// TIA Portal project "BackUp" (V15)

(* hardware
DEVICE "S7-1200 station_1"  S7-1200 Station
   slot 0: "Rack_0"  S7-1200 Rack  Rack  V1.0
   slot 1: "PLC_1"  CPU 1214C DC/DC/DC  6ES7 214-1AG40-0XB0  V4.2
   slot 2: "DQ 8x24VDC _1"  SM 1222 DQ8 x 24VDC  6ES7 222-1BF32-0XB0  V2.0
*)

// ===== PLC "PLC_1"  CPU 1214C DC/DC/DC =====

VAR_GLOBAL   // PLC tag table "Tabla de variables estándar"
   "Ready" AT %I0.2 : Bool;
   "INP/ABSB0" AT %I0.0 : Bool;
   "ZSP/ABSB1" AT %I0.1 : Bool;
   "TLC/ABST Trans. Data Ready M" AT %I0.3 : Bool;
   "Alarm" AT %I0.4 : Bool;
   "SENSOR BOT LEFT" AT %I0.7 : Bool;
   "SENSOR BOT MID" AT %I0.6 : Bool;
   "SENSOR BOT RIGHT" AT %I0.5 : Bool;
   "SENSOR TOP LEFT" AT %I1.0 : Bool;
   "SENSOR TOP MID" AT %I1.1 : Bool;
   "SENSOR TOP RIGHT" AT %I1.2 : Bool;
   "SENSOR VERT TOP" AT %I1.3 : Bool;
   "SENSOR OPT. DOOR" AT %I1.5 : Bool;
   "SENSOR VERT BOT" AT %I1.4 : Bool;
   "Magnetic Brake" AT %Q8.6 : Bool;
   "Clear" AT %Q0.2 : Bool;
   "Axis_1_Pulse" AT %Q0.0 : Bool;
   "Axis_1_Direction" AT %Q0.1 : Bool;
   "PC/ABSM Transfer Mode" AT %Q0.3 : Bool;
   "TL/ABSR Request" AT %Q0.4 : Bool;
   "Son" AT %Q0.5 : Bool;
   "BOT. PNEU. ACT. RIGHT" AT %Q0.7 : Bool;
   "Lasers ON" AT %Q8.2 : Bool;
   "Lasers Zero 1" AT %Q8.3 : Bool;
   "Lasers Zero 2" AT %Q8.4 : Bool;
   "Lasers Zero 3" AT %Q8.5 : Bool;
   "PNEU. ACT. DOWN" AT %Q8.0 : Bool;
   "PNEU. ACT. UP" AT %Q8.1 : Bool;
   "BOT. PNEU. ACT. LEFT" AT %Q0.6 : Bool;
   "TOP. PNEU. ACT. LEFT" AT %Q1.0 : Bool;
   "TOP. PNEU. ACT. RIGHT" AT %Q1.1 : Bool;
   "Pilot Valve" AT %Q8.7 : Bool;
   "Magnetic Brake M" AT %M101.0 : Bool;
   "Set Home Axis" AT %M101.1 : Bool;
   "TL/ABSR Request M" AT %M0.3 : Bool;
   "PC/ABSM Transfer Mode M" AT %M0.2 : Bool;
   "Son M" AT %M101.2 : Bool;
   "INP/ABSB0 M" AT %M1.0 : Bool;
   "ZSP/ABSB1 M" AT %M1.1 : Bool;
   "TLC/ABST Trans. Data Ready" AT %M1.2 : Bool;
   "Step-0" AT %M5.0 : Bool;
   "Step-1" AT %M5.1 : Bool;
   "System_Byte" AT %MB3 : Byte;
   "FirstScan" AT %M3.0 : Bool;
   "DiagStatusUpdate" AT %M3.1 : Bool;
   "AlwaysTRUE" AT %M3.2 : Bool;
   "AlwaysFALSE" AT %M3.3 : Bool;
   "Step-2" AT %M5.2 : Bool;
   "Step-3" AT %M5.3 : Bool;
   "Step-4" AT %M5.4 : Bool;
   "Step-5" AT %M5.5 : Bool;
   "Step-6" AT %M5.6 : Bool;
   "Step-7" AT %M5.7 : Bool;
   "Step-8" AT %M6.0 : Bool;
   "Step-9" AT %M6.1 : Bool;
   "Step-10" AT %M6.2 : Bool;
   "Step-11" AT %M6.3 : Bool;
   "Step-12" AT %M6.4 : Bool;
   "Step-13" AT %M6.5 : Bool;
   "Step-14" AT %M6.6 : Bool;
   "Step-15" AT %M6.7 : Bool;
   "Step-16" AT %M7.0 : Bool;
   "Step-17" AT %M7.1 : Bool;
   "Step-18" AT %M7.2 : Bool;
   "Step-19" AT %M7.3 : Bool;
   "Step-20" AT %M7.4 : Bool;
   "Step-21" AT %M7.5 : Bool;
   "Step-22" AT %M7.6 : Bool;
   "Step-23" AT %M7.7 : Bool;
   "Step-24" AT %M8.0 : Bool;
   "Step-25" AT %M8.1 : Bool;
   "Step-26" AT %M8.2 : Bool;
   "Step-27" AT %M8.3 : Bool;
   "Step-28" AT %M8.4 : Bool;
   "Step-29" AT %M8.5 : Bool;
   "Step-30" AT %M8.6 : Bool;
   "Step-31" AT %M8.7 : Bool;
   "Step-32" AT %M9.0 : Bool;
   "Step-33" AT %M9.1 : Bool;
   "Step-34" AT %M9.2 : Bool;
   "Step-35" AT %M9.3 : Bool;
   "Step-36" AT %M9.4 : Bool;
   "Step-37" AT %M9.5 : Bool;
   "Step-38" AT %M9.6 : Bool;
   "Step-39" AT %M9.7 : Bool;
   "Step-40" AT %M10.0 : Bool;
   "Checksum OK" AT %M0.6 : Bool;
   "Step-41" AT %M10.1 : Bool;
   "Checksum M" AT %M0.7 : Bool;
   "Tranfer Mode Bit" AT %M1.3 : Bool;
   "Bit 25" AT %M11.0 : Bool;
   "Bit 26" AT %M11.1 : Bool;
   "Bit 27" AT %M11.2 : Bool;
   "Bit 28" AT %M11.3 : Bool;
   "Bit 29" AT %M11.4 : Bool;
   "Bit 30" AT %M11.5 : Bool;
   "Bit 31" AT %M11.6 : Bool;
   "Bit 32" AT %M11.7 : Bool;
   "Bit 17" AT %M12.0 : Bool;
   "Bit 18" AT %M12.1 : Bool;
   "Bit 19" AT %M12.2 : Bool;
   "Bit 20" AT %M12.3 : Bool;
   "Bit 21" AT %M12.4 : Bool;
   "Bit 22" AT %M12.5 : Bool;
   "Bit 23" AT %M12.6 : Bool;
   "Bit 24" AT %M12.7 : Bool;
   "Bit 9" AT %M13.0 : Bool;
   "Bit 10" AT %M13.1 : Bool;
   "Bit 11" AT %M13.2 : Bool;
   "Bit 12" AT %M13.3 : Bool;
   "Bit 13" AT %M13.4 : Bool;
   "Bit 14" AT %M13.5 : Bool;
   "Bit 15" AT %M13.6 : Bool;
   "Bit 16" AT %M13.7 : Bool;
   "Bit 1" AT %M14.0 : Bool;
   "Bit 2" AT %M14.1 : Bool;
   "Bit 3" AT %M14.2 : Bool;
   "Bit 4" AT %M14.3 : Bool;
   "Bit 5" AT %M14.4 : Bool;
   "Bit 6" AT %M14.5 : Bool;
   "Bit 7" AT %M14.6 : Bool;
   "Bit 8" AT %M14.7 : Bool;
   "Bit 1 Checksum" AT %M30.0 : Bool;
   "Bit 2 Checksum" AT %M30.1 : Bool;
   "Bit 3 Checksum" AT %M30.2 : Bool;
   "Bit 4 Checksum" AT %M30.3 : Bool;
   "Bit 5 Checksum" AT %M30.4 : Bool;
   "Bit 6 Checksum" AT %M30.5 : Bool;
   "ABS DoubleWord" AT %MD11 : DWord;
   "ABS DoubleInteger" AT %MD16 : DInt;
   "Checksum Byte" AT %MB30 : Byte;
   "Checksum Integer" AT %MW40 : Int;
   "Reset ABM Transfer" AT %M1.4 : Bool;
   "Step-42" AT %M10.2 : Bool;
   "Enable Axis" AT %M1.5 : Bool;
   "Move Absolute" AT %M101.3 : Bool;
   "Position" AT %MD42 : Real;
   "Velocity" AT %MD46 : Real;
   "Jog Back" AT %M101.4 : Bool;
   "Jog Forw" AT %M101.6 : Bool;
   "Jog" AT %M2.1 : Bool;
   "Home" AT %M2.2 : Bool;
   "Move Relative" AT %M101.7 : Bool;
   "BOT. PNEU. AUT. START" AT %M100.7 : Bool;
   "Lasers ON M" AT %M100.0 : Bool;
   "Lasers Zero 1 M" AT %M100.1 : Bool;
   "Lasers Zero 2 M" AT %M100.2 : Bool;
   "Lasers Zero 3 M" AT %M100.3 : Bool;
   "Home PLC" AT %M101.5 : Bool;
   "Home Done" AT %M138.0 : Bool;
   "Ramp Down" AT %MD50 : Real;
   "Ramp Up" AT %MD54 : Real;
   "Execute Ramp" AT %M103.0 : Bool;
   "Halt" AT %M103.1 : Bool;
   "BOT. PNEU. ACT. RIGHT M" AT %M100.5 : Bool;
   "BOT. PNEU. ACT. LEFT M" AT %M100.6 : Bool;
   "VELOCITY REAL" AT %MD700 : Real;
   "MB VELOCITY 2" AT %MW105 : UInt;
   "RAMP DOWN REAL" AT %MD704 : Real;
   "RAMP UP REAL" AT %MD708 : Real;
   "MB RAMP DOWN 2" AT %MW107 : UInt;
   "MB RAMP UP 2" AT %MW109 : UInt;
   "MB VELOCITY 1" AT %MW104 : UInt;
   "MB RAMP DOWN 1" AT %MW106 : UInt;
   "MB RAMP UP 1" AT %MW108 : UInt;
   "MB POSITION 1" AT %MW110 : UInt;
   "MB POSITION 2" AT %MW112 : UInt;
   "MB POSITION" AT %MD114 : DWord;
   "POSITION REAL" AT %MD118 : DInt;
   "Tag_4" AT %MW114 : UInt;
   "Tag_1" AT %MW116 : UInt;
   "PLC POSITION" AT %MD122 : Real;
   "PLC POS 1" AT %MW130 : UInt;
   "PLC POS 2" AT %MW132 : UInt;
   "PLC POS MULT" AT %MD126 : DInt;
   "PLC POS DW" AT %MD130 : DWord;
   "ABS POS" AT %MD134 : DWord;
   "Tag_2" AT %M500.0 : Bool;
   "Tag_3" AT %M500.1 : Bool;
   "Tag_5" AT %M500.2 : Bool;
   "Tag_6" AT %M400.0 : Bool;
   "HOME PNEU. ACT." AT %M100.4 : Bool;
   "Tag_8" AT %M400.1 : Bool;
   "Tag_9" AT %M500.6 : Bool;
   "Tag_10" AT %M500.4 : Bool;
   "Tag_11" AT %M500.5 : Bool;
   "Tag_12" AT %M500.3 : Bool;
   "Tag_13" AT %M501.0 : Bool;
   "Tag_14" AT %M501.1 : Bool;
   "Tag_15" AT %M501.2 : Bool;
   "Tag_16" AT %M501.3 : Bool;
   "Tag_17" AT %M501.4 : Bool;
   "Tag_18" AT %M501.5 : Bool;
   "Tag_19" AT %M501.6 : Bool;
   "Tag_20" AT %M501.7 : Bool;
   "Tag_21" AT %M502.0 : Bool;
   "Bot. Act. Mid. Pos." AT %M138.1 : Bool;
   "Bot. Act. Rig. Pos." AT %M138.2 : Bool;
   "TOP. PNEU. ACT. RIGHT M" AT %M103.2 : Bool;
   "TOP. PNEU. ACT. LEFT M" AT %M103.3 : Bool;
   "HEAD PNEU. ACT. DOWN" AT %M103.4 : Bool;
   "HEAD PNEU. ACT. UP" AT %M103.5 : Bool;
   "Tag_22" AT %M503.0 : Bool;
   "Tag_23" AT %M503.2 : Bool;
   "Tag_24" AT %M503.4 : Bool;
   "Tag_25" AT %M503.6 : Bool;
   "Tag_26" AT %M503.1 : Bool;
   "Tag_27" AT %M503.5 : Bool;
   "Tag_28" AT %M503.3 : Bool;
   "Tag_29" AT %M504.0 : Bool;
   "Tag_30" AT %M504.1 : Bool;
   "Tag_31" AT %M505.0 : Bool;
   "Tag_32" AT %M504.2 : Bool;
   "Tag_33" AT %M504.3 : Bool;
   "Tag_34" AT %M504.4 : Bool;
   "Tag_35" AT %M504.5 : Bool;
   "Tag_36" AT %M504.6 : Bool;
   "Tag_37" AT %M504.7 : Bool;
   "TOP. PNEU. AUT. START" AT %M103.6 : Bool;
   "Top Act. Mid. Pos." AT %M138.3 : Bool;
   "Top Act. Rig. Pos." AT %M138.4 : Bool;
   "Tag_7" AT %M506.0 : Bool;
   "Tag_38" AT %M506.1 : Bool;
   "Tag_39" AT %M506.2 : Bool;
   "Tag_40" AT %M506.3 : Bool;
   "Tag_41" AT %M506.4 : Bool;
   "HOME VERT. PNE. ACT." AT %M103.7 : Bool;
   "AUTO VERT. PNE. ACT." AT %M102.0 : Bool;
   "Tag_42" AT %M507.0 : Bool;
   "Tag_43" AT %M507.1 : Bool;
   "Tag_44" AT %M507.2 : Bool;
   "Tag_45" AT %M507.4 : Bool;
   "Tag_46" AT %M507.3 : Bool;
   "Tag_47" AT %M507.5 : Bool;
   "Door In Pos." AT %M138.5 : Bool;
   "Door Out Pos" AT %M138.6 : Bool;
   "Home Door" AT %M138.7 : Bool;
   "Tag_48" AT %M507.6 : Bool;
   "Pilot Valve M" AT %M102.1 : Bool;
   "Tag_49" AT %M503.7 : Bool;
   "Tag_50" AT %M500.7 : Bool;
   "Tag_51" AT %M505.1 : Bool;
   "Tag_52" AT %M502.1 : Bool;
END_VAR

DATA_BLOCK "MBConfig"   // DB13
{ S7_Optimized_Access := 'TRUE' }
VERSION : 0.1
   VAR
      CONNECT : TCON_IP_v4;
      NDR : Bool;
      DR : Bool;
      ERROR : Bool;
      STATE : Word;
   END_VAR
BEGIN
   CONNECT.InterfaceId := 64;
   CONNECT.ID := 1;
   CONNECT.ConnectionType := 11;
   CONNECT.RemoteAddress.ADDR[1] := 192;
   CONNECT.RemoteAddress.ADDR[2] := 168;
   CONNECT.RemoteAddress.ADDR[3] := 0;
   CONNECT.RemoteAddress.ADDR[4] := 101;
   CONNECT.LocalPort := 502;
END_DATA_BLOCK

DATA_BLOCK "BUFF"   // DB14
{ S7_Optimized_Access := 'TRUE' }
VERSION : 0.1
   VAR
      DATA : Array[0..100] of Word;
   END_VAR
BEGIN
END_DATA_BLOCK

DATA_BLOCK "RETAIN MEMORY"   // DB16
{ S7_Optimized_Access := 'TRUE' }
VERSION : 0.1
   VAR RETAIN
      SBLR : Bool;
      SBMR : Bool;
      SBRR : Bool;
      STLR : Bool;
      STMR : Bool;
      STRR : Bool;
      SVTR : Bool;
      SVBR : Bool;
   END_VAR
BEGIN
END_DATA_BLOCK

// folder: System blocks/Program resources

DATA_BLOCK "IEC_Timer_0_DB"   // DB2
{ S7_Optimized_Access := 'TRUE' }
AUTHOR : Simatic
FAMILY : IEC
NAME : IEC_TMR
VERSION : 1.0
// stored: InstanceOfName IEC_TIMER
"IEC_TIMER"
BEGIN
END_DATA_BLOCK

DATA_BLOCK "IEC_Timer_0_DB_1"   // DB3
{ S7_Optimized_Access := 'TRUE' }
AUTHOR : Simatic
FAMILY : IEC
NAME : IEC_TMR
VERSION : 1.0
// stored: InstanceOfName IEC_TIMER
"IEC_TIMER"
BEGIN
END_DATA_BLOCK

DATA_BLOCK "IEC_Timer_0_DB_3"   // DB5
{ S7_Optimized_Access := 'TRUE' }
AUTHOR : Simatic
FAMILY : IEC
NAME : IEC_TMR
VERSION : 1.0
// stored: InstanceOfName IEC_TIMER
"IEC_TIMER"
BEGIN
END_DATA_BLOCK

DATA_BLOCK "IEC_Timer_0_DB_2"   // DB15
{ S7_Optimized_Access := 'TRUE' }
AUTHOR : Simatic
FAMILY : IEC
NAME : IEC_TMR
VERSION : 1.0
// stored: InstanceOfName IEC_TIMER
"IEC_TIMER"
BEGIN
END_DATA_BLOCK

DATA_BLOCK "IEC_Timer_0_DB_4"   // DB17
{ S7_Optimized_Access := 'TRUE' }
AUTHOR : Simatic
FAMILY : IEC
NAME : IEC_TMR
VERSION : 1.0
// stored: InstanceOfName IEC_TIMER
"IEC_TIMER"
BEGIN
END_DATA_BLOCK

DATA_BLOCK "IEC_Timer_0_DB_5"   // DB18
{ S7_Optimized_Access := 'TRUE' }
AUTHOR : Simatic
FAMILY : IEC
NAME : IEC_TMR
VERSION : 1.0
// stored: InstanceOfName IEC_TIMER
"IEC_TIMER"
BEGIN
END_DATA_BLOCK

DATA_BLOCK "IEC_Timer_0_DB_6"   // DB19
{ S7_Optimized_Access := 'TRUE' }
AUTHOR : Simatic
FAMILY : IEC
NAME : IEC_TMR
VERSION : 1.0
// stored: InstanceOfName IEC_TIMER
"IEC_TIMER"
BEGIN
END_DATA_BLOCK

DATA_BLOCK "IEC_Timer_0_DB_7"   // DB20
{ S7_Optimized_Access := 'TRUE' }
AUTHOR : Simatic
FAMILY : IEC
NAME : IEC_TMR
VERSION : 1.0
// stored: InstanceOfName IEC_TIMER
"IEC_TIMER"
BEGIN
END_DATA_BLOCK

// folder: (top level)

DATA_BLOCK "Axis_1"   // DB1, Motion_DB
{ S7_Optimized_Access := 'TRUE' }
AUTHOR : SIMATIC
FAMILY : BasicMC
NAME : TO_PosAx
VERSION : 5.0
// stored: InstanceOfName TO_PositioningAxis
"TO_PositioningAxis"
BEGIN
   // Axis.LengthUnitNormalized.Distance = 1013
   // Axis.ReadyInput_AddressCU = %M3.2
   // Axis.OnlinePtoModeCU = 16#0000_0002
   // Axis.DirectionOutputEnabledCU = TRUE
   // Axis.SelectedChannel2EnumCU = %Q0.1
   // Axis.SelectedChannel1EnumCU = %Q0.0
   // Pulse.MinDeltaDeltaFrequencyCU = 0.004
   // Pulse.MaxDeltaDeltaFrequencyCU = 1.0E+10
   // Pulse.MinDeltaFrequencyCU = 0.005
   // Pulse.MaxDeltaFrequencyCU = 9.5E+9
   // Pulse.MinFrequencyCU = 1.0
   // Pulse.MaxFrequencyCU = 100000.0
   // Pulse.OutputSourceCU = 16#0000_0000
   // Axis.SelectPTO = 0
END_DATA_BLOCK

FUNCTION "GRAFCET ABS" : Void   // FC1, LAD
{ S7_Optimized_Access := 'TRUE' }
VERSION : 0.1
BEGIN

REGION Network 1
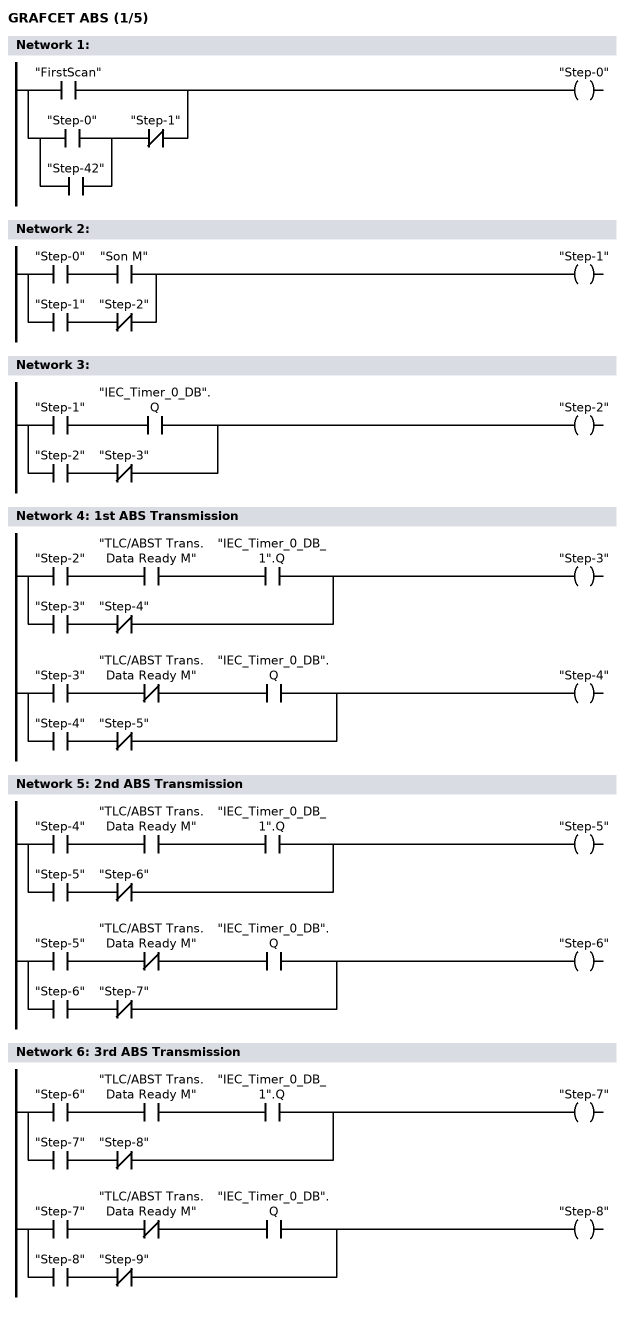
   RUNG wire#powerrail
      Contact( "FirstScan" )
      wire#w1
      Coil( "Step-0" )
   END_RUNG
   RUNG wire#powerrail
      Contact( "Step-0" )
      wire#w2
      I_Contact( "Step-1" )
   END_RUNG wire#w1
   RUNG wire#powerrail
      Contact( "Step-42" )
   END_RUNG wire#w2
   // the same network as SCL:
   "Step-0" := "FirstScan" OR (("Step-0" OR "Step-42") AND NOT "Step-1");
END_REGION

REGION Network 2
   RUNG wire#powerrail
      Contact( "Step-0" )
      Contact( "Son M" )
      wire#w1
      Coil( "Step-1" )
   END_RUNG
   RUNG wire#powerrail
      Contact( "Step-1" )
      I_Contact( "Step-2" )
   END_RUNG wire#w1
   // the same network as SCL:
   "Step-1" := ("Step-0" AND "Son M") OR ("Step-1" AND NOT "Step-2");
END_REGION

REGION Network 3
   RUNG wire#powerrail
      Contact( "Step-1" )
      Contact( "IEC_Timer_0_DB".Q )
      wire#w1
      Coil( "Step-2" )
   END_RUNG
   RUNG wire#powerrail
      Contact( "Step-2" )
      I_Contact( "Step-3" )
   END_RUNG wire#w1
   // the same network as SCL:
   "Step-2" := ("Step-1" AND "IEC_Timer_0_DB".Q) OR ("Step-2" AND NOT "Step-3");
END_REGION

REGION Network 4: 1st ABS Transmission
   RUNG wire#powerrail
      Contact( "Step-2" )
      Contact( "TLC/ABST Trans. Data Ready M" )
      Contact( "IEC_Timer_0_DB_1".Q )
      wire#w1
      Coil( "Step-3" )
   END_RUNG
   RUNG wire#powerrail
      Contact( "Step-3" )
      I_Contact( "Step-4" )
   END_RUNG wire#w1
   RUNG wire#powerrail
      Contact( "Step-3" )
      I_Contact( "TLC/ABST Trans. Data Ready M" )
      Contact( "IEC_Timer_0_DB".Q )
      wire#w2
      Coil( "Step-4" )
   END_RUNG
   RUNG wire#powerrail
      Contact( "Step-4" )
      I_Contact( "Step-5" )
   END_RUNG wire#w2
   // the same network as SCL:
   "Step-3" := ("Step-2" AND "TLC/ABST Trans. Data Ready M" AND "IEC_Timer_0_DB_1".Q) OR ("Step-3" AND NOT "Step-4");
   "Step-4" := ("Step-3" AND NOT "TLC/ABST Trans. Data Ready M" AND "IEC_Timer_0_DB".Q) OR ("Step-4" AND NOT "Step-5");
END_REGION

REGION Network 5: 2nd ABS Transmission
   RUNG wire#powerrail
      Contact( "Step-4" )
      Contact( "TLC/ABST Trans. Data Ready M" )
      Contact( "IEC_Timer_0_DB_1".Q )
      wire#w1
      Coil( "Step-5" )
   END_RUNG
   RUNG wire#powerrail
      Contact( "Step-5" )
      I_Contact( "Step-6" )
   END_RUNG wire#w1
   RUNG wire#powerrail
      Contact( "Step-5" )
      I_Contact( "TLC/ABST Trans. Data Ready M" )
      Contact( "IEC_Timer_0_DB".Q )
      wire#w2
      Coil( "Step-6" )
   END_RUNG
   RUNG wire#powerrail
      Contact( "Step-6" )
      I_Contact( "Step-7" )
   END_RUNG wire#w2
   // the same network as SCL:
   "Step-5" := ("Step-4" AND "TLC/ABST Trans. Data Ready M" AND "IEC_Timer_0_DB_1".Q) OR ("Step-5" AND NOT "Step-6");
   "Step-6" := ("Step-5" AND NOT "TLC/ABST Trans. Data Ready M" AND "IEC_Timer_0_DB".Q) OR ("Step-6" AND NOT "Step-7");
END_REGION

REGION Network 6: 3rd ABS Transmission
   RUNG wire#powerrail
      Contact( "Step-6" )
      Contact( "TLC/ABST Trans. Data Ready M" )
      Contact( "IEC_Timer_0_DB_1".Q )
      wire#w1
      Coil( "Step-7" )
   END_RUNG
   RUNG wire#powerrail
      Contact( "Step-7" )
      I_Contact( "Step-8" )
   END_RUNG wire#w1
   RUNG wire#powerrail
      Contact( "Step-7" )
      I_Contact( "TLC/ABST Trans. Data Ready M" )
      Contact( "IEC_Timer_0_DB".Q )
      wire#w2
      Coil( "Step-8" )
   END_RUNG
   RUNG wire#powerrail
      Contact( "Step-8" )
      I_Contact( "Step-9" )
   END_RUNG wire#w2
   // the same network as SCL:
   "Step-7" := ("Step-6" AND "TLC/ABST Trans. Data Ready M" AND "IEC_Timer_0_DB_1".Q) OR ("Step-7" AND NOT "Step-8");
   "Step-8" := ("Step-7" AND NOT "TLC/ABST Trans. Data Ready M" AND "IEC_Timer_0_DB".Q) OR ("Step-8" AND NOT "Step-9");
END_REGION

REGION Network 7: 4th ABS Transmission
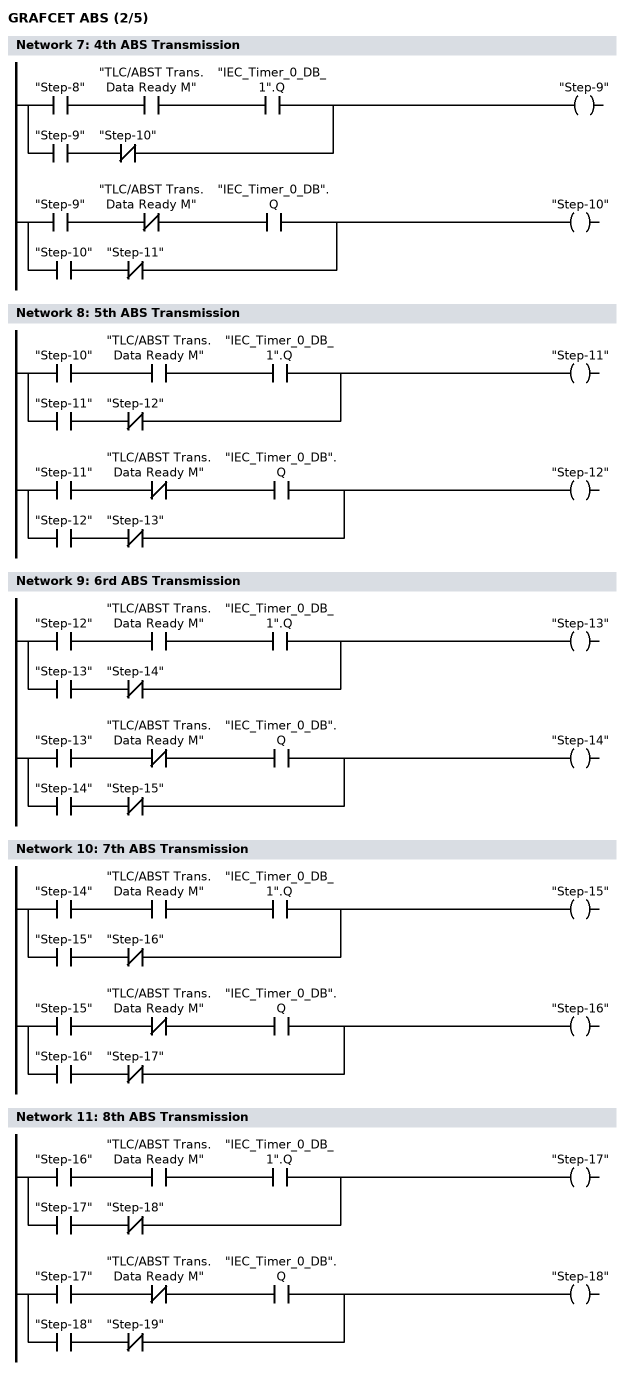
   RUNG wire#powerrail
      Contact( "Step-8" )
      Contact( "TLC/ABST Trans. Data Ready M" )
      Contact( "IEC_Timer_0_DB_1".Q )
      wire#w1
      Coil( "Step-9" )
   END_RUNG
   RUNG wire#powerrail
      Contact( "Step-9" )
      I_Contact( "Step-10" )
   END_RUNG wire#w1
   RUNG wire#powerrail
      Contact( "Step-9" )
      I_Contact( "TLC/ABST Trans. Data Ready M" )
      Contact( "IEC_Timer_0_DB".Q )
      wire#w2
      Coil( "Step-10" )
   END_RUNG
   RUNG wire#powerrail
      Contact( "Step-10" )
      I_Contact( "Step-11" )
   END_RUNG wire#w2
   // the same network as SCL:
   "Step-9" := ("Step-8" AND "TLC/ABST Trans. Data Ready M" AND "IEC_Timer_0_DB_1".Q) OR ("Step-9" AND NOT "Step-10");
   "Step-10" := ("Step-9" AND NOT "TLC/ABST Trans. Data Ready M" AND "IEC_Timer_0_DB".Q) OR ("Step-10" AND NOT "Step-11");
END_REGION

REGION Network 8: 5th ABS Transmission
   RUNG wire#powerrail
      Contact( "Step-10" )
      Contact( "TLC/ABST Trans. Data Ready M" )
      Contact( "IEC_Timer_0_DB_1".Q )
      wire#w1
      Coil( "Step-11" )
   END_RUNG
   RUNG wire#powerrail
      Contact( "Step-11" )
      I_Contact( "Step-12" )
   END_RUNG wire#w1
   RUNG wire#powerrail
      Contact( "Step-11" )
      I_Contact( "TLC/ABST Trans. Data Ready M" )
      Contact( "IEC_Timer_0_DB".Q )
      wire#w2
      Coil( "Step-12" )
   END_RUNG
   RUNG wire#powerrail
      Contact( "Step-12" )
      I_Contact( "Step-13" )
   END_RUNG wire#w2
   // the same network as SCL:
   "Step-11" := ("Step-10" AND "TLC/ABST Trans. Data Ready M" AND "IEC_Timer_0_DB_1".Q) OR ("Step-11" AND NOT "Step-12");
   "Step-12" := ("Step-11" AND NOT "TLC/ABST Trans. Data Ready M" AND "IEC_Timer_0_DB".Q) OR ("Step-12" AND NOT "Step-13");
END_REGION

REGION Network 9: 6rd ABS Transmission
   RUNG wire#powerrail
      Contact( "Step-12" )
      Contact( "TLC/ABST Trans. Data Ready M" )
      Contact( "IEC_Timer_0_DB_1".Q )
      wire#w1
      Coil( "Step-13" )
   END_RUNG
   RUNG wire#powerrail
      Contact( "Step-13" )
      I_Contact( "Step-14" )
   END_RUNG wire#w1
   RUNG wire#powerrail
      Contact( "Step-13" )
      I_Contact( "TLC/ABST Trans. Data Ready M" )
      Contact( "IEC_Timer_0_DB".Q )
      wire#w2
      Coil( "Step-14" )
   END_RUNG
   RUNG wire#powerrail
      Contact( "Step-14" )
      I_Contact( "Step-15" )
   END_RUNG wire#w2
   // the same network as SCL:
   "Step-13" := ("Step-12" AND "TLC/ABST Trans. Data Ready M" AND "IEC_Timer_0_DB_1".Q) OR ("Step-13" AND NOT "Step-14");
   "Step-14" := ("Step-13" AND NOT "TLC/ABST Trans. Data Ready M" AND "IEC_Timer_0_DB".Q) OR ("Step-14" AND NOT "Step-15");
END_REGION

REGION Network 10: 7th ABS Transmission
   RUNG wire#powerrail
      Contact( "Step-14" )
      Contact( "TLC/ABST Trans. Data Ready M" )
      Contact( "IEC_Timer_0_DB_1".Q )
      wire#w1
      Coil( "Step-15" )
   END_RUNG
   RUNG wire#powerrail
      Contact( "Step-15" )
      I_Contact( "Step-16" )
   END_RUNG wire#w1
   RUNG wire#powerrail
      Contact( "Step-15" )
      I_Contact( "TLC/ABST Trans. Data Ready M" )
      Contact( "IEC_Timer_0_DB".Q )
      wire#w2
      Coil( "Step-16" )
   END_RUNG
   RUNG wire#powerrail
      Contact( "Step-16" )
      I_Contact( "Step-17" )
   END_RUNG wire#w2
   // the same network as SCL:
   "Step-15" := ("Step-14" AND "TLC/ABST Trans. Data Ready M" AND "IEC_Timer_0_DB_1".Q) OR ("Step-15" AND NOT "Step-16");
   "Step-16" := ("Step-15" AND NOT "TLC/ABST Trans. Data Ready M" AND "IEC_Timer_0_DB".Q) OR ("Step-16" AND NOT "Step-17");
END_REGION

REGION Network 11: 8th ABS Transmission
   RUNG wire#powerrail
      Contact( "Step-16" )
      Contact( "TLC/ABST Trans. Data Ready M" )
      Contact( "IEC_Timer_0_DB_1".Q )
      wire#w1
      Coil( "Step-17" )
   END_RUNG
   RUNG wire#powerrail
      Contact( "Step-17" )
      I_Contact( "Step-18" )
   END_RUNG wire#w1
   RUNG wire#powerrail
      Contact( "Step-17" )
      I_Contact( "TLC/ABST Trans. Data Ready M" )
      Contact( "IEC_Timer_0_DB".Q )
      wire#w2
      Coil( "Step-18" )
   END_RUNG
   RUNG wire#powerrail
      Contact( "Step-18" )
      I_Contact( "Step-19" )
   END_RUNG wire#w2
   // the same network as SCL:
   "Step-17" := ("Step-16" AND "TLC/ABST Trans. Data Ready M" AND "IEC_Timer_0_DB_1".Q) OR ("Step-17" AND NOT "Step-18");
   "Step-18" := ("Step-17" AND NOT "TLC/ABST Trans. Data Ready M" AND "IEC_Timer_0_DB".Q) OR ("Step-18" AND NOT "Step-19");
END_REGION

REGION Network 12: 9th ABS Transmission
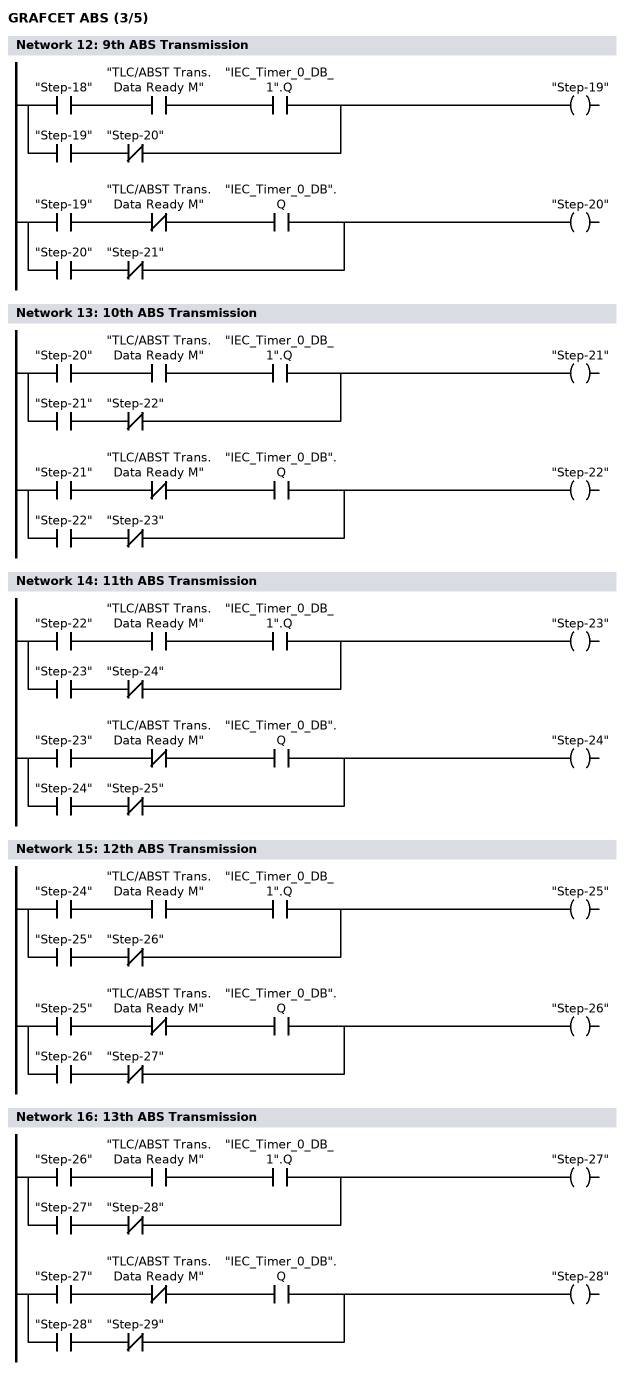
   RUNG wire#powerrail
      Contact( "Step-18" )
      Contact( "TLC/ABST Trans. Data Ready M" )
      Contact( "IEC_Timer_0_DB_1".Q )
      wire#w1
      Coil( "Step-19" )
   END_RUNG
   RUNG wire#powerrail
      Contact( "Step-19" )
      I_Contact( "Step-20" )
   END_RUNG wire#w1
   RUNG wire#powerrail
      Contact( "Step-19" )
      I_Contact( "TLC/ABST Trans. Data Ready M" )
      Contact( "IEC_Timer_0_DB".Q )
      wire#w2
      Coil( "Step-20" )
   END_RUNG
   RUNG wire#powerrail
      Contact( "Step-20" )
      I_Contact( "Step-21" )
   END_RUNG wire#w2
   // the same network as SCL:
   "Step-19" := ("Step-18" AND "TLC/ABST Trans. Data Ready M" AND "IEC_Timer_0_DB_1".Q) OR ("Step-19" AND NOT "Step-20");
   "Step-20" := ("Step-19" AND NOT "TLC/ABST Trans. Data Ready M" AND "IEC_Timer_0_DB".Q) OR ("Step-20" AND NOT "Step-21");
END_REGION

REGION Network 13: 10th ABS Transmission
   RUNG wire#powerrail
      Contact( "Step-20" )
      Contact( "TLC/ABST Trans. Data Ready M" )
      Contact( "IEC_Timer_0_DB_1".Q )
      wire#w1
      Coil( "Step-21" )
   END_RUNG
   RUNG wire#powerrail
      Contact( "Step-21" )
      I_Contact( "Step-22" )
   END_RUNG wire#w1
   RUNG wire#powerrail
      Contact( "Step-21" )
      I_Contact( "TLC/ABST Trans. Data Ready M" )
      Contact( "IEC_Timer_0_DB".Q )
      wire#w2
      Coil( "Step-22" )
   END_RUNG
   RUNG wire#powerrail
      Contact( "Step-22" )
      I_Contact( "Step-23" )
   END_RUNG wire#w2
   // the same network as SCL:
   "Step-21" := ("Step-20" AND "TLC/ABST Trans. Data Ready M" AND "IEC_Timer_0_DB_1".Q) OR ("Step-21" AND NOT "Step-22");
   "Step-22" := ("Step-21" AND NOT "TLC/ABST Trans. Data Ready M" AND "IEC_Timer_0_DB".Q) OR ("Step-22" AND NOT "Step-23");
END_REGION

REGION Network 14: 11th ABS Transmission
   RUNG wire#powerrail
      Contact( "Step-22" )
      Contact( "TLC/ABST Trans. Data Ready M" )
      Contact( "IEC_Timer_0_DB_1".Q )
      wire#w1
      Coil( "Step-23" )
   END_RUNG
   RUNG wire#powerrail
      Contact( "Step-23" )
      I_Contact( "Step-24" )
   END_RUNG wire#w1
   RUNG wire#powerrail
      Contact( "Step-23" )
      I_Contact( "TLC/ABST Trans. Data Ready M" )
      Contact( "IEC_Timer_0_DB".Q )
      wire#w2
      Coil( "Step-24" )
   END_RUNG
   RUNG wire#powerrail
      Contact( "Step-24" )
      I_Contact( "Step-25" )
   END_RUNG wire#w2
   // the same network as SCL:
   "Step-23" := ("Step-22" AND "TLC/ABST Trans. Data Ready M" AND "IEC_Timer_0_DB_1".Q) OR ("Step-23" AND NOT "Step-24");
   "Step-24" := ("Step-23" AND NOT "TLC/ABST Trans. Data Ready M" AND "IEC_Timer_0_DB".Q) OR ("Step-24" AND NOT "Step-25");
END_REGION

REGION Network 15: 12th ABS Transmission
   RUNG wire#powerrail
      Contact( "Step-24" )
      Contact( "TLC/ABST Trans. Data Ready M" )
      Contact( "IEC_Timer_0_DB_1".Q )
      wire#w1
      Coil( "Step-25" )
   END_RUNG
   RUNG wire#powerrail
      Contact( "Step-25" )
      I_Contact( "Step-26" )
   END_RUNG wire#w1
   RUNG wire#powerrail
      Contact( "Step-25" )
      I_Contact( "TLC/ABST Trans. Data Ready M" )
      Contact( "IEC_Timer_0_DB".Q )
      wire#w2
      Coil( "Step-26" )
   END_RUNG
   RUNG wire#powerrail
      Contact( "Step-26" )
      I_Contact( "Step-27" )
   END_RUNG wire#w2
   // the same network as SCL:
   "Step-25" := ("Step-24" AND "TLC/ABST Trans. Data Ready M" AND "IEC_Timer_0_DB_1".Q) OR ("Step-25" AND NOT "Step-26");
   "Step-26" := ("Step-25" AND NOT "TLC/ABST Trans. Data Ready M" AND "IEC_Timer_0_DB".Q) OR ("Step-26" AND NOT "Step-27");
END_REGION

REGION Network 16: 13th ABS Transmission
   RUNG wire#powerrail
      Contact( "Step-26" )
      Contact( "TLC/ABST Trans. Data Ready M" )
      Contact( "IEC_Timer_0_DB_1".Q )
      wire#w1
      Coil( "Step-27" )
   END_RUNG
   RUNG wire#powerrail
      Contact( "Step-27" )
      I_Contact( "Step-28" )
   END_RUNG wire#w1
   RUNG wire#powerrail
      Contact( "Step-27" )
      I_Contact( "TLC/ABST Trans. Data Ready M" )
      Contact( "IEC_Timer_0_DB".Q )
      wire#w2
      Coil( "Step-28" )
   END_RUNG
   RUNG wire#powerrail
      Contact( "Step-28" )
      I_Contact( "Step-29" )
   END_RUNG wire#w2
   // the same network as SCL:
   "Step-27" := ("Step-26" AND "TLC/ABST Trans. Data Ready M" AND "IEC_Timer_0_DB_1".Q) OR ("Step-27" AND NOT "Step-28");
   "Step-28" := ("Step-27" AND NOT "TLC/ABST Trans. Data Ready M" AND "IEC_Timer_0_DB".Q) OR ("Step-28" AND NOT "Step-29");
END_REGION

REGION Network 17: 14th ABS Transmission
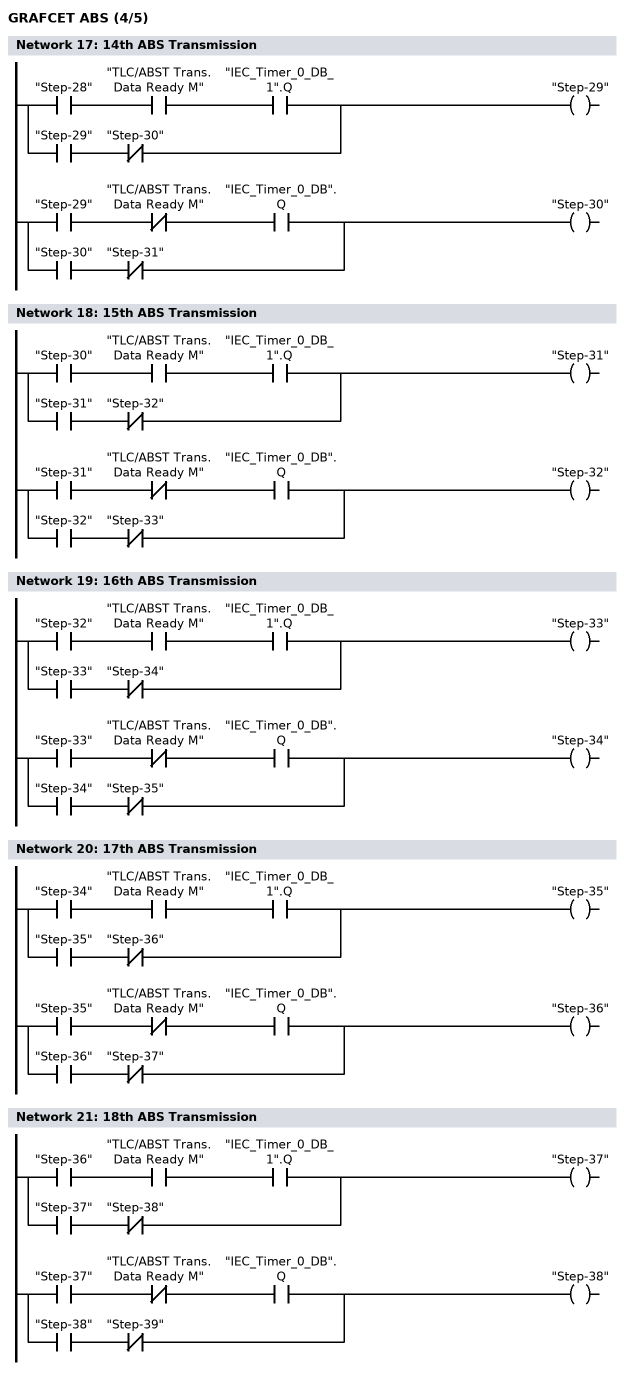
   RUNG wire#powerrail
      Contact( "Step-28" )
      Contact( "TLC/ABST Trans. Data Ready M" )
      Contact( "IEC_Timer_0_DB_1".Q )
      wire#w1
      Coil( "Step-29" )
   END_RUNG
   RUNG wire#powerrail
      Contact( "Step-29" )
      I_Contact( "Step-30" )
   END_RUNG wire#w1
   RUNG wire#powerrail
      Contact( "Step-29" )
      I_Contact( "TLC/ABST Trans. Data Ready M" )
      Contact( "IEC_Timer_0_DB".Q )
      wire#w2
      Coil( "Step-30" )
   END_RUNG
   RUNG wire#powerrail
      Contact( "Step-30" )
      I_Contact( "Step-31" )
   END_RUNG wire#w2
   // the same network as SCL:
   "Step-29" := ("Step-28" AND "TLC/ABST Trans. Data Ready M" AND "IEC_Timer_0_DB_1".Q) OR ("Step-29" AND NOT "Step-30");
   "Step-30" := ("Step-29" AND NOT "TLC/ABST Trans. Data Ready M" AND "IEC_Timer_0_DB".Q) OR ("Step-30" AND NOT "Step-31");
END_REGION

REGION Network 18: 15th ABS Transmission
   RUNG wire#powerrail
      Contact( "Step-30" )
      Contact( "TLC/ABST Trans. Data Ready M" )
      Contact( "IEC_Timer_0_DB_1".Q )
      wire#w1
      Coil( "Step-31" )
   END_RUNG
   RUNG wire#powerrail
      Contact( "Step-31" )
      I_Contact( "Step-32" )
   END_RUNG wire#w1
   RUNG wire#powerrail
      Contact( "Step-31" )
      I_Contact( "TLC/ABST Trans. Data Ready M" )
      Contact( "IEC_Timer_0_DB".Q )
      wire#w2
      Coil( "Step-32" )
   END_RUNG
   RUNG wire#powerrail
      Contact( "Step-32" )
      I_Contact( "Step-33" )
   END_RUNG wire#w2
   // the same network as SCL:
   "Step-31" := ("Step-30" AND "TLC/ABST Trans. Data Ready M" AND "IEC_Timer_0_DB_1".Q) OR ("Step-31" AND NOT "Step-32");
   "Step-32" := ("Step-31" AND NOT "TLC/ABST Trans. Data Ready M" AND "IEC_Timer_0_DB".Q) OR ("Step-32" AND NOT "Step-33");
END_REGION

REGION Network 19: 16th ABS Transmission
   RUNG wire#powerrail
      Contact( "Step-32" )
      Contact( "TLC/ABST Trans. Data Ready M" )
      Contact( "IEC_Timer_0_DB_1".Q )
      wire#w1
      Coil( "Step-33" )
   END_RUNG
   RUNG wire#powerrail
      Contact( "Step-33" )
      I_Contact( "Step-34" )
   END_RUNG wire#w1
   RUNG wire#powerrail
      Contact( "Step-33" )
      I_Contact( "TLC/ABST Trans. Data Ready M" )
      Contact( "IEC_Timer_0_DB".Q )
      wire#w2
      Coil( "Step-34" )
   END_RUNG
   RUNG wire#powerrail
      Contact( "Step-34" )
      I_Contact( "Step-35" )
   END_RUNG wire#w2
   // the same network as SCL:
   "Step-33" := ("Step-32" AND "TLC/ABST Trans. Data Ready M" AND "IEC_Timer_0_DB_1".Q) OR ("Step-33" AND NOT "Step-34");
   "Step-34" := ("Step-33" AND NOT "TLC/ABST Trans. Data Ready M" AND "IEC_Timer_0_DB".Q) OR ("Step-34" AND NOT "Step-35");
END_REGION

REGION Network 20: 17th ABS Transmission
   RUNG wire#powerrail
      Contact( "Step-34" )
      Contact( "TLC/ABST Trans. Data Ready M" )
      Contact( "IEC_Timer_0_DB_1".Q )
      wire#w1
      Coil( "Step-35" )
   END_RUNG
   RUNG wire#powerrail
      Contact( "Step-35" )
      I_Contact( "Step-36" )
   END_RUNG wire#w1
   RUNG wire#powerrail
      Contact( "Step-35" )
      I_Contact( "TLC/ABST Trans. Data Ready M" )
      Contact( "IEC_Timer_0_DB".Q )
      wire#w2
      Coil( "Step-36" )
   END_RUNG
   RUNG wire#powerrail
      Contact( "Step-36" )
      I_Contact( "Step-37" )
   END_RUNG wire#w2
   // the same network as SCL:
   "Step-35" := ("Step-34" AND "TLC/ABST Trans. Data Ready M" AND "IEC_Timer_0_DB_1".Q) OR ("Step-35" AND NOT "Step-36");
   "Step-36" := ("Step-35" AND NOT "TLC/ABST Trans. Data Ready M" AND "IEC_Timer_0_DB".Q) OR ("Step-36" AND NOT "Step-37");
END_REGION

REGION Network 21: 18th ABS Transmission
   RUNG wire#powerrail
      Contact( "Step-36" )
      Contact( "TLC/ABST Trans. Data Ready M" )
      Contact( "IEC_Timer_0_DB_1".Q )
      wire#w1
      Coil( "Step-37" )
   END_RUNG
   RUNG wire#powerrail
      Contact( "Step-37" )
      I_Contact( "Step-38" )
   END_RUNG wire#w1
   RUNG wire#powerrail
      Contact( "Step-37" )
      I_Contact( "TLC/ABST Trans. Data Ready M" )
      Contact( "IEC_Timer_0_DB".Q )
      wire#w2
      Coil( "Step-38" )
   END_RUNG
   RUNG wire#powerrail
      Contact( "Step-38" )
      I_Contact( "Step-39" )
   END_RUNG wire#w2
   // the same network as SCL:
   "Step-37" := ("Step-36" AND "TLC/ABST Trans. Data Ready M" AND "IEC_Timer_0_DB_1".Q) OR ("Step-37" AND NOT "Step-38");
   "Step-38" := ("Step-37" AND NOT "TLC/ABST Trans. Data Ready M" AND "IEC_Timer_0_DB".Q) OR ("Step-38" AND NOT "Step-39");
END_REGION

REGION Network 22: 19th ABS Transmission
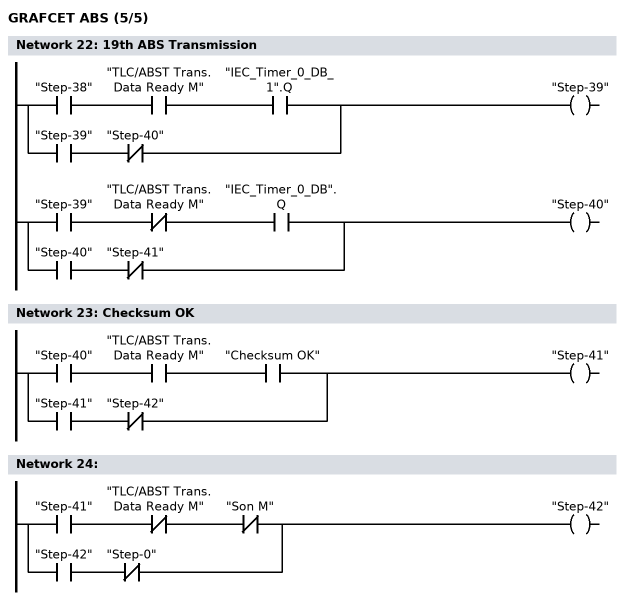
   RUNG wire#powerrail
      Contact( "Step-38" )
      Contact( "TLC/ABST Trans. Data Ready M" )
      Contact( "IEC_Timer_0_DB_1".Q )
      wire#w1
      Coil( "Step-39" )
   END_RUNG
   RUNG wire#powerrail
      Contact( "Step-39" )
      I_Contact( "Step-40" )
   END_RUNG wire#w1
   RUNG wire#powerrail
      Contact( "Step-39" )
      I_Contact( "TLC/ABST Trans. Data Ready M" )
      Contact( "IEC_Timer_0_DB".Q )
      wire#w2
      Coil( "Step-40" )
   END_RUNG
   RUNG wire#powerrail
      Contact( "Step-40" )
      I_Contact( "Step-41" )
   END_RUNG wire#w2
   // the same network as SCL:
   "Step-39" := ("Step-38" AND "TLC/ABST Trans. Data Ready M" AND "IEC_Timer_0_DB_1".Q) OR ("Step-39" AND NOT "Step-40");
   "Step-40" := ("Step-39" AND NOT "TLC/ABST Trans. Data Ready M" AND "IEC_Timer_0_DB".Q) OR ("Step-40" AND NOT "Step-41");
END_REGION

REGION Network 23: Checksum OK
   RUNG wire#powerrail
      Contact( "Step-40" )
      Contact( "TLC/ABST Trans. Data Ready M" )
      Contact( "Checksum OK" )
      wire#w1
      Coil( "Step-41" )
   END_RUNG
   RUNG wire#powerrail
      Contact( "Step-41" )
      I_Contact( "Step-42" )
   END_RUNG wire#w1
   // the same network as SCL:
   "Step-41" := ("Step-40" AND "TLC/ABST Trans. Data Ready M" AND "Checksum OK") OR ("Step-41" AND NOT "Step-42");
END_REGION

REGION Network 24
   RUNG wire#powerrail
      Contact( "Step-41" )
      I_Contact( "TLC/ABST Trans. Data Ready M" )
      I_Contact( "Son M" )
      wire#w1
      Coil( "Step-42" )
   END_RUNG
   RUNG wire#powerrail
      Contact( "Step-42" )
      I_Contact( "Step-0" )
   END_RUNG wire#w1
   // the same network as SCL:
   "Step-42" := ("Step-41" AND NOT "TLC/ABST Trans. Data Ready M" AND NOT "Son M") OR ("Step-42" AND NOT "Step-0");
END_REGION
END_FUNCTION

FUNCTION "OUTPUT GRAFCET ABS" : Void   // FC2, LAD
{ S7_Optimized_Access := 'TRUE' }
VERSION : 0.1
   VAR_TEMP   // added for the SCL form of the ladder/FBD networks
      _w1 : Bool;
   END_VAR
BEGIN

REGION Network 1
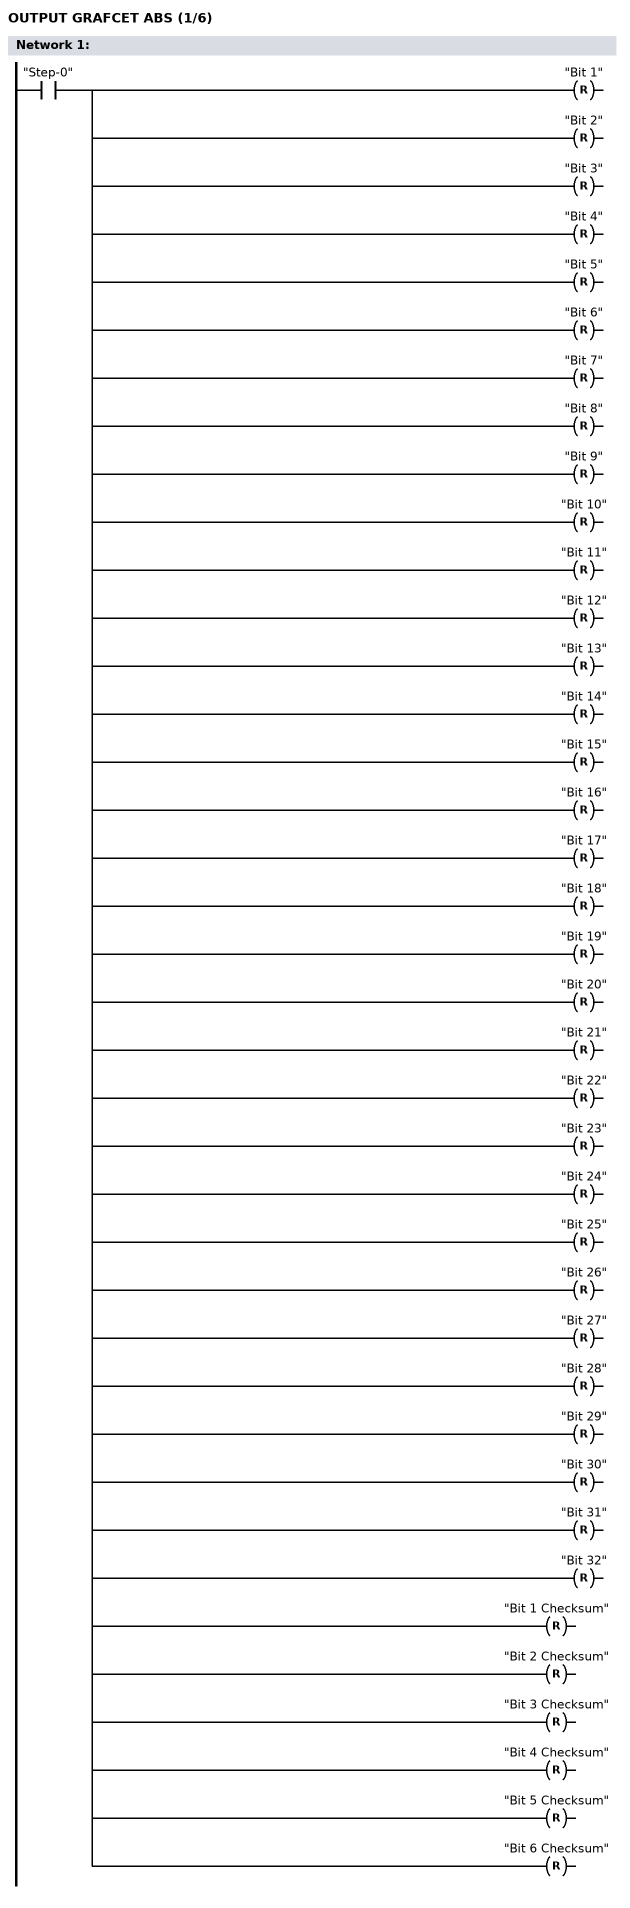
   RUNG wire#powerrail
      Contact( "Step-0" )
      wire#w1
      R_Coil( "Bit 1" )
   END_RUNG
   RUNG wire#w1
      R_Coil( "Bit 2" )
   END_RUNG
   RUNG wire#w1
      R_Coil( "Bit 3" )
   END_RUNG
   RUNG wire#w1
      R_Coil( "Bit 4" )
   END_RUNG
   RUNG wire#w1
      R_Coil( "Bit 5" )
   END_RUNG
   RUNG wire#w1
      R_Coil( "Bit 6" )
   END_RUNG
   RUNG wire#w1
      R_Coil( "Bit 7" )
   END_RUNG
   RUNG wire#w1
      R_Coil( "Bit 8" )
   END_RUNG
   RUNG wire#w1
      R_Coil( "Bit 9" )
   END_RUNG
   RUNG wire#w1
      R_Coil( "Bit 10" )
   END_RUNG
   RUNG wire#w1
      R_Coil( "Bit 11" )
   END_RUNG
   RUNG wire#w1
      R_Coil( "Bit 12" )
   END_RUNG
   RUNG wire#w1
      R_Coil( "Bit 13" )
   END_RUNG
   RUNG wire#w1
      R_Coil( "Bit 14" )
   END_RUNG
   RUNG wire#w1
      R_Coil( "Bit 15" )
   END_RUNG
   RUNG wire#w1
      R_Coil( "Bit 16" )
   END_RUNG
   RUNG wire#w1
      R_Coil( "Bit 17" )
   END_RUNG
   RUNG wire#w1
      R_Coil( "Bit 18" )
   END_RUNG
   RUNG wire#w1
      R_Coil( "Bit 19" )
   END_RUNG
   RUNG wire#w1
      R_Coil( "Bit 20" )
   END_RUNG
   RUNG wire#w1
      R_Coil( "Bit 21" )
   END_RUNG
   RUNG wire#w1
      R_Coil( "Bit 22" )
   END_RUNG
   RUNG wire#w1
      R_Coil( "Bit 23" )
   END_RUNG
   RUNG wire#w1
      R_Coil( "Bit 24" )
   END_RUNG
   RUNG wire#w1
      R_Coil( "Bit 25" )
   END_RUNG
   RUNG wire#w1
      R_Coil( "Bit 26" )
   END_RUNG
   RUNG wire#w1
      R_Coil( "Bit 27" )
   END_RUNG
   RUNG wire#w1
      R_Coil( "Bit 28" )
   END_RUNG
   RUNG wire#w1
      R_Coil( "Bit 29" )
   END_RUNG
   RUNG wire#w1
      R_Coil( "Bit 30" )
   END_RUNG
   RUNG wire#w1
      R_Coil( "Bit 31" )
   END_RUNG
   RUNG wire#w1
      R_Coil( "Bit 32" )
   END_RUNG
   RUNG wire#w1
      R_Coil( "Bit 1 Checksum" )
   END_RUNG
   RUNG wire#w1
      R_Coil( "Bit 2 Checksum" )
   END_RUNG
   RUNG wire#w1
      R_Coil( "Bit 3 Checksum" )
   END_RUNG
   RUNG wire#w1
      R_Coil( "Bit 4 Checksum" )
   END_RUNG
   RUNG wire#w1
      R_Coil( "Bit 5 Checksum" )
   END_RUNG
   RUNG wire#w1
      R_Coil( "Bit 6 Checksum" )
   END_RUNG
   // the same network as SCL:
   IF "Step-0" THEN
       "Bit 1" := FALSE;
       "Bit 2" := FALSE;
       "Bit 3" := FALSE;
       "Bit 4" := FALSE;
       "Bit 5" := FALSE;
       "Bit 6" := FALSE;
       "Bit 7" := FALSE;
       "Bit 8" := FALSE;
       "Bit 9" := FALSE;
       "Bit 10" := FALSE;
       "Bit 11" := FALSE;
       "Bit 12" := FALSE;
       "Bit 13" := FALSE;
       "Bit 14" := FALSE;
       "Bit 15" := FALSE;
       "Bit 16" := FALSE;
       "Bit 17" := FALSE;
       "Bit 18" := FALSE;
       "Bit 19" := FALSE;
       "Bit 20" := FALSE;
       "Bit 21" := FALSE;
       "Bit 22" := FALSE;
       "Bit 23" := FALSE;
       "Bit 24" := FALSE;
       "Bit 25" := FALSE;
       "Bit 26" := FALSE;
       "Bit 27" := FALSE;
       "Bit 28" := FALSE;
       "Bit 29" := FALSE;
       "Bit 30" := FALSE;
       "Bit 31" := FALSE;
       "Bit 32" := FALSE;
       "Bit 1 Checksum" := FALSE;
       "Bit 2 Checksum" := FALSE;
       "Bit 3 Checksum" := FALSE;
       "Bit 4 Checksum" := FALSE;
       "Bit 5 Checksum" := FALSE;
       "Bit 6 Checksum" := FALSE;
   END_IF;
END_REGION

REGION Network 2: Step-1
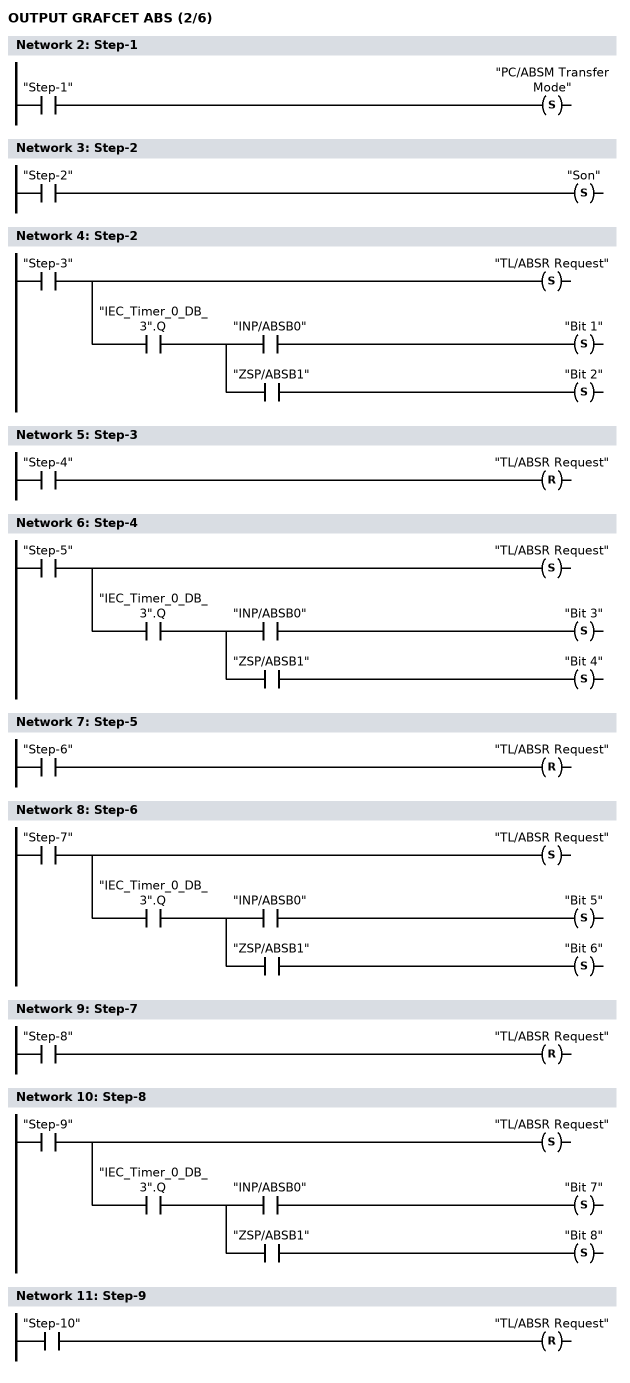
   RUNG wire#powerrail
      Contact( "Step-1" )
      S_Coil( "PC/ABSM Transfer Mode" )
   END_RUNG
   // the same network as SCL:
   IF "Step-1" THEN "PC/ABSM Transfer Mode" := TRUE; END_IF;
END_REGION

REGION Network 3: Step-2
   RUNG wire#powerrail
      Contact( "Step-2" )
      S_Coil( "Son" )
   END_RUNG
   // the same network as SCL:
   IF "Step-2" THEN "Son" := TRUE; END_IF;
END_REGION

REGION Network 4: Step-2
   RUNG wire#powerrail
      Contact( "Step-3" )
      wire#w1
      S_Coil( "TL/ABSR Request" )
   END_RUNG
   RUNG wire#w1
      Contact( "IEC_Timer_0_DB_3".Q )
      wire#w2
      Contact( "INP/ABSB0" )
      S_Coil( "Bit 1" )
   END_RUNG
   RUNG wire#w2
      Contact( "ZSP/ABSB1" )
      S_Coil( "Bit 2" )
   END_RUNG
   // the same network as SCL:
   IF "Step-3" THEN "TL/ABSR Request" := TRUE; END_IF;
   #_w1 := "Step-3" AND "IEC_Timer_0_DB_3".Q;
   IF #_w1 AND "INP/ABSB0" THEN "Bit 1" := TRUE; END_IF;
   IF #_w1 AND "ZSP/ABSB1" THEN "Bit 2" := TRUE; END_IF;
END_REGION

REGION Network 5: Step-3
   RUNG wire#powerrail
      Contact( "Step-4" )
      R_Coil( "TL/ABSR Request" )
   END_RUNG
   // the same network as SCL:
   IF "Step-4" THEN "TL/ABSR Request" := FALSE; END_IF;
END_REGION

REGION Network 6: Step-4
   RUNG wire#powerrail
      Contact( "Step-5" )
      wire#w1
      S_Coil( "TL/ABSR Request" )
   END_RUNG
   RUNG wire#w1
      Contact( "IEC_Timer_0_DB_3".Q )
      wire#w2
      Contact( "INP/ABSB0" )
      S_Coil( "Bit 3" )
   END_RUNG
   RUNG wire#w2
      Contact( "ZSP/ABSB1" )
      S_Coil( "Bit 4" )
   END_RUNG
   // the same network as SCL:
   IF "Step-5" THEN "TL/ABSR Request" := TRUE; END_IF;
   #_w1 := "Step-5" AND "IEC_Timer_0_DB_3".Q;
   IF #_w1 AND "INP/ABSB0" THEN "Bit 3" := TRUE; END_IF;
   IF #_w1 AND "ZSP/ABSB1" THEN "Bit 4" := TRUE; END_IF;
END_REGION

REGION Network 7: Step-5
   RUNG wire#powerrail
      Contact( "Step-6" )
      R_Coil( "TL/ABSR Request" )
   END_RUNG
   // the same network as SCL:
   IF "Step-6" THEN "TL/ABSR Request" := FALSE; END_IF;
END_REGION

REGION Network 8: Step-6
   RUNG wire#powerrail
      Contact( "Step-7" )
      wire#w1
      S_Coil( "TL/ABSR Request" )
   END_RUNG
   RUNG wire#w1
      Contact( "IEC_Timer_0_DB_3".Q )
      wire#w2
      Contact( "INP/ABSB0" )
      S_Coil( "Bit 5" )
   END_RUNG
   RUNG wire#w2
      Contact( "ZSP/ABSB1" )
      S_Coil( "Bit 6" )
   END_RUNG
   // the same network as SCL:
   IF "Step-7" THEN "TL/ABSR Request" := TRUE; END_IF;
   #_w1 := "Step-7" AND "IEC_Timer_0_DB_3".Q;
   IF #_w1 AND "INP/ABSB0" THEN "Bit 5" := TRUE; END_IF;
   IF #_w1 AND "ZSP/ABSB1" THEN "Bit 6" := TRUE; END_IF;
END_REGION

REGION Network 9: Step-7
   RUNG wire#powerrail
      Contact( "Step-8" )
      R_Coil( "TL/ABSR Request" )
   END_RUNG
   // the same network as SCL:
   IF "Step-8" THEN "TL/ABSR Request" := FALSE; END_IF;
END_REGION

REGION Network 10: Step-8
   RUNG wire#powerrail
      Contact( "Step-9" )
      wire#w1
      S_Coil( "TL/ABSR Request" )
   END_RUNG
   RUNG wire#w1
      Contact( "IEC_Timer_0_DB_3".Q )
      wire#w2
      Contact( "INP/ABSB0" )
      S_Coil( "Bit 7" )
   END_RUNG
   RUNG wire#w2
      Contact( "ZSP/ABSB1" )
      S_Coil( "Bit 8" )
   END_RUNG
   // the same network as SCL:
   IF "Step-9" THEN "TL/ABSR Request" := TRUE; END_IF;
   #_w1 := "Step-9" AND "IEC_Timer_0_DB_3".Q;
   IF #_w1 AND "INP/ABSB0" THEN "Bit 7" := TRUE; END_IF;
   IF #_w1 AND "ZSP/ABSB1" THEN "Bit 8" := TRUE; END_IF;
END_REGION

REGION Network 11: Step-9
   RUNG wire#powerrail
      Contact( "Step-10" )
      R_Coil( "TL/ABSR Request" )
   END_RUNG
   // the same network as SCL:
   IF "Step-10" THEN "TL/ABSR Request" := FALSE; END_IF;
END_REGION

REGION Network 12: Step-10
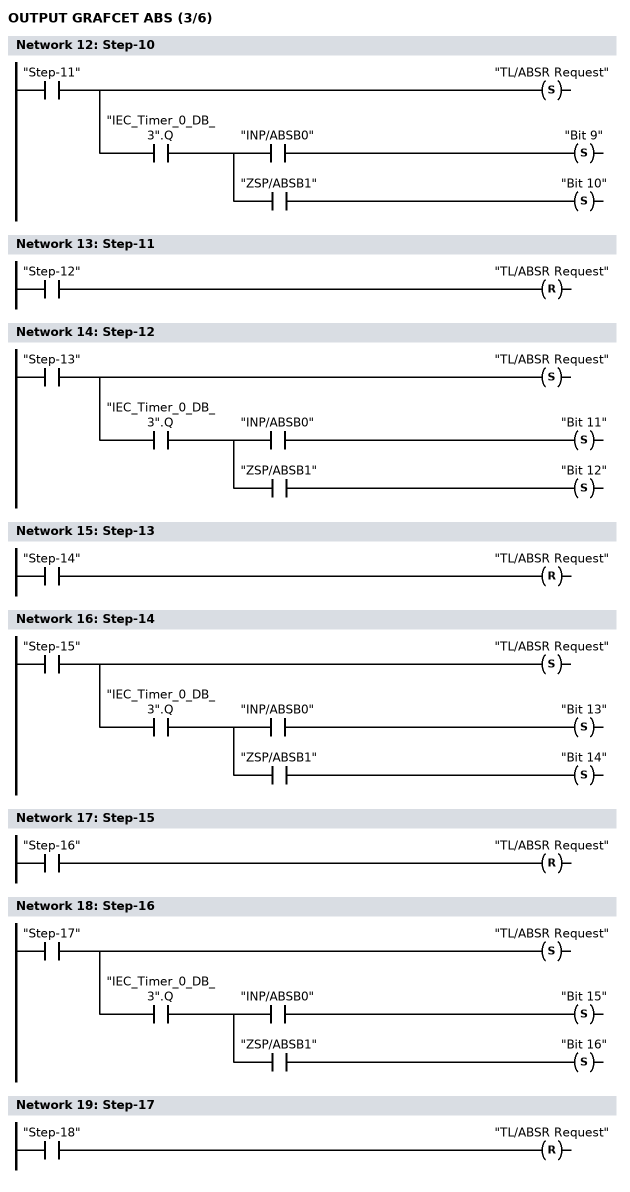
   RUNG wire#powerrail
      Contact( "Step-11" )
      wire#w1
      S_Coil( "TL/ABSR Request" )
   END_RUNG
   RUNG wire#w1
      Contact( "IEC_Timer_0_DB_3".Q )
      wire#w2
      Contact( "INP/ABSB0" )
      S_Coil( "Bit 9" )
   END_RUNG
   RUNG wire#w2
      Contact( "ZSP/ABSB1" )
      S_Coil( "Bit 10" )
   END_RUNG
   // the same network as SCL:
   IF "Step-11" THEN "TL/ABSR Request" := TRUE; END_IF;
   #_w1 := "Step-11" AND "IEC_Timer_0_DB_3".Q;
   IF #_w1 AND "INP/ABSB0" THEN "Bit 9" := TRUE; END_IF;
   IF #_w1 AND "ZSP/ABSB1" THEN "Bit 10" := TRUE; END_IF;
END_REGION

REGION Network 13: Step-11
   RUNG wire#powerrail
      Contact( "Step-12" )
      R_Coil( "TL/ABSR Request" )
   END_RUNG
   // the same network as SCL:
   IF "Step-12" THEN "TL/ABSR Request" := FALSE; END_IF;
END_REGION

REGION Network 14: Step-12
   RUNG wire#powerrail
      Contact( "Step-13" )
      wire#w1
      S_Coil( "TL/ABSR Request" )
   END_RUNG
   RUNG wire#w1
      Contact( "IEC_Timer_0_DB_3".Q )
      wire#w2
      Contact( "INP/ABSB0" )
      S_Coil( "Bit 11" )
   END_RUNG
   RUNG wire#w2
      Contact( "ZSP/ABSB1" )
      S_Coil( "Bit 12" )
   END_RUNG
   // the same network as SCL:
   IF "Step-13" THEN "TL/ABSR Request" := TRUE; END_IF;
   #_w1 := "Step-13" AND "IEC_Timer_0_DB_3".Q;
   IF #_w1 AND "INP/ABSB0" THEN "Bit 11" := TRUE; END_IF;
   IF #_w1 AND "ZSP/ABSB1" THEN "Bit 12" := TRUE; END_IF;
END_REGION

REGION Network 15: Step-13
   RUNG wire#powerrail
      Contact( "Step-14" )
      R_Coil( "TL/ABSR Request" )
   END_RUNG
   // the same network as SCL:
   IF "Step-14" THEN "TL/ABSR Request" := FALSE; END_IF;
END_REGION

REGION Network 16: Step-14
   RUNG wire#powerrail
      Contact( "Step-15" )
      wire#w1
      S_Coil( "TL/ABSR Request" )
   END_RUNG
   RUNG wire#w1
      Contact( "IEC_Timer_0_DB_3".Q )
      wire#w2
      Contact( "INP/ABSB0" )
      S_Coil( "Bit 13" )
   END_RUNG
   RUNG wire#w2
      Contact( "ZSP/ABSB1" )
      S_Coil( "Bit 14" )
   END_RUNG
   // the same network as SCL:
   IF "Step-15" THEN "TL/ABSR Request" := TRUE; END_IF;
   #_w1 := "Step-15" AND "IEC_Timer_0_DB_3".Q;
   IF #_w1 AND "INP/ABSB0" THEN "Bit 13" := TRUE; END_IF;
   IF #_w1 AND "ZSP/ABSB1" THEN "Bit 14" := TRUE; END_IF;
END_REGION

REGION Network 17: Step-15
   RUNG wire#powerrail
      Contact( "Step-16" )
      R_Coil( "TL/ABSR Request" )
   END_RUNG
   // the same network as SCL:
   IF "Step-16" THEN "TL/ABSR Request" := FALSE; END_IF;
END_REGION

REGION Network 18: Step-16
   RUNG wire#powerrail
      Contact( "Step-17" )
      wire#w1
      S_Coil( "TL/ABSR Request" )
   END_RUNG
   RUNG wire#w1
      Contact( "IEC_Timer_0_DB_3".Q )
      wire#w2
      Contact( "INP/ABSB0" )
      S_Coil( "Bit 15" )
   END_RUNG
   RUNG wire#w2
      Contact( "ZSP/ABSB1" )
      S_Coil( "Bit 16" )
   END_RUNG
   // the same network as SCL:
   IF "Step-17" THEN "TL/ABSR Request" := TRUE; END_IF;
   #_w1 := "Step-17" AND "IEC_Timer_0_DB_3".Q;
   IF #_w1 AND "INP/ABSB0" THEN "Bit 15" := TRUE; END_IF;
   IF #_w1 AND "ZSP/ABSB1" THEN "Bit 16" := TRUE; END_IF;
END_REGION

REGION Network 19: Step-17
   RUNG wire#powerrail
      Contact( "Step-18" )
      R_Coil( "TL/ABSR Request" )
   END_RUNG
   // the same network as SCL:
   IF "Step-18" THEN "TL/ABSR Request" := FALSE; END_IF;
END_REGION

REGION Network 20: Step-18
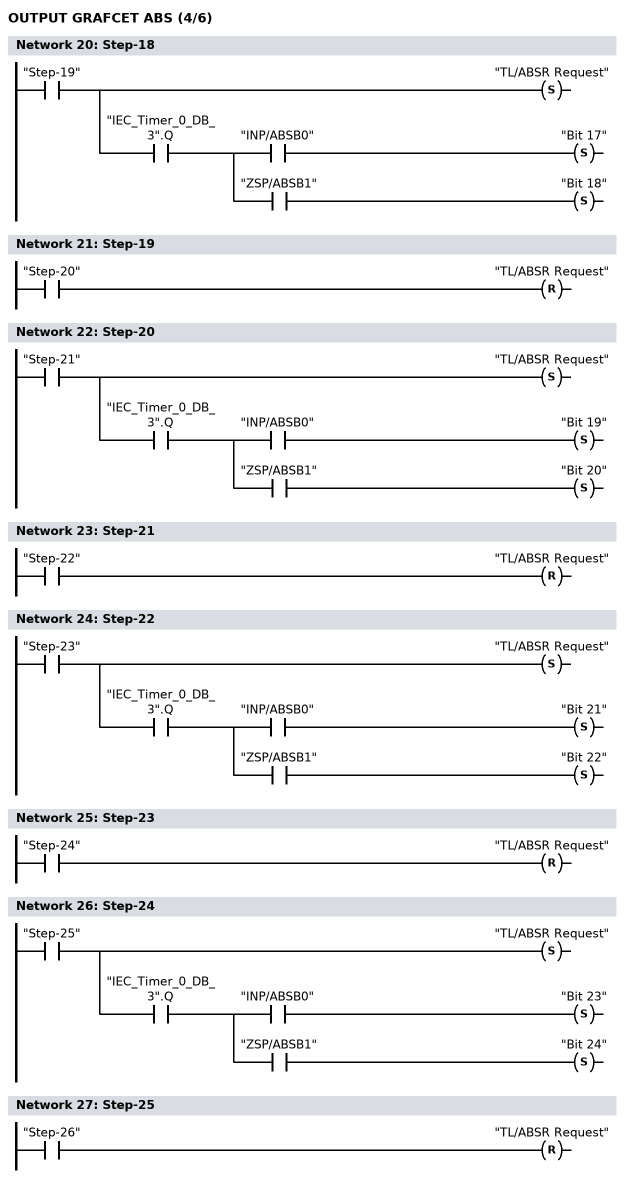
   RUNG wire#powerrail
      Contact( "Step-19" )
      wire#w1
      S_Coil( "TL/ABSR Request" )
   END_RUNG
   RUNG wire#w1
      Contact( "IEC_Timer_0_DB_3".Q )
      wire#w2
      Contact( "INP/ABSB0" )
      S_Coil( "Bit 17" )
   END_RUNG
   RUNG wire#w2
      Contact( "ZSP/ABSB1" )
      S_Coil( "Bit 18" )
   END_RUNG
   // the same network as SCL:
   IF "Step-19" THEN "TL/ABSR Request" := TRUE; END_IF;
   #_w1 := "Step-19" AND "IEC_Timer_0_DB_3".Q;
   IF #_w1 AND "INP/ABSB0" THEN "Bit 17" := TRUE; END_IF;
   IF #_w1 AND "ZSP/ABSB1" THEN "Bit 18" := TRUE; END_IF;
END_REGION

REGION Network 21: Step-19
   RUNG wire#powerrail
      Contact( "Step-20" )
      R_Coil( "TL/ABSR Request" )
   END_RUNG
   // the same network as SCL:
   IF "Step-20" THEN "TL/ABSR Request" := FALSE; END_IF;
END_REGION

REGION Network 22: Step-20
   RUNG wire#powerrail
      Contact( "Step-21" )
      wire#w1
      S_Coil( "TL/ABSR Request" )
   END_RUNG
   RUNG wire#w1
      Contact( "IEC_Timer_0_DB_3".Q )
      wire#w2
      Contact( "INP/ABSB0" )
      S_Coil( "Bit 19" )
   END_RUNG
   RUNG wire#w2
      Contact( "ZSP/ABSB1" )
      S_Coil( "Bit 20" )
   END_RUNG
   // the same network as SCL:
   IF "Step-21" THEN "TL/ABSR Request" := TRUE; END_IF;
   #_w1 := "Step-21" AND "IEC_Timer_0_DB_3".Q;
   IF #_w1 AND "INP/ABSB0" THEN "Bit 19" := TRUE; END_IF;
   IF #_w1 AND "ZSP/ABSB1" THEN "Bit 20" := TRUE; END_IF;
END_REGION

REGION Network 23: Step-21
   RUNG wire#powerrail
      Contact( "Step-22" )
      R_Coil( "TL/ABSR Request" )
   END_RUNG
   // the same network as SCL:
   IF "Step-22" THEN "TL/ABSR Request" := FALSE; END_IF;
END_REGION

REGION Network 24: Step-22
   RUNG wire#powerrail
      Contact( "Step-23" )
      wire#w1
      S_Coil( "TL/ABSR Request" )
   END_RUNG
   RUNG wire#w1
      Contact( "IEC_Timer_0_DB_3".Q )
      wire#w2
      Contact( "INP/ABSB0" )
      S_Coil( "Bit 21" )
   END_RUNG
   RUNG wire#w2
      Contact( "ZSP/ABSB1" )
      S_Coil( "Bit 22" )
   END_RUNG
   // the same network as SCL:
   IF "Step-23" THEN "TL/ABSR Request" := TRUE; END_IF;
   #_w1 := "Step-23" AND "IEC_Timer_0_DB_3".Q;
   IF #_w1 AND "INP/ABSB0" THEN "Bit 21" := TRUE; END_IF;
   IF #_w1 AND "ZSP/ABSB1" THEN "Bit 22" := TRUE; END_IF;
END_REGION

REGION Network 25: Step-23
   RUNG wire#powerrail
      Contact( "Step-24" )
      R_Coil( "TL/ABSR Request" )
   END_RUNG
   // the same network as SCL:
   IF "Step-24" THEN "TL/ABSR Request" := FALSE; END_IF;
END_REGION

REGION Network 26: Step-24
   RUNG wire#powerrail
      Contact( "Step-25" )
      wire#w1
      S_Coil( "TL/ABSR Request" )
   END_RUNG
   RUNG wire#w1
      Contact( "IEC_Timer_0_DB_3".Q )
      wire#w2
      Contact( "INP/ABSB0" )
      S_Coil( "Bit 23" )
   END_RUNG
   RUNG wire#w2
      Contact( "ZSP/ABSB1" )
      S_Coil( "Bit 24" )
   END_RUNG
   // the same network as SCL:
   IF "Step-25" THEN "TL/ABSR Request" := TRUE; END_IF;
   #_w1 := "Step-25" AND "IEC_Timer_0_DB_3".Q;
   IF #_w1 AND "INP/ABSB0" THEN "Bit 23" := TRUE; END_IF;
   IF #_w1 AND "ZSP/ABSB1" THEN "Bit 24" := TRUE; END_IF;
END_REGION

REGION Network 27: Step-25
   RUNG wire#powerrail
      Contact( "Step-26" )
      R_Coil( "TL/ABSR Request" )
   END_RUNG
   // the same network as SCL:
   IF "Step-26" THEN "TL/ABSR Request" := FALSE; END_IF;
END_REGION

REGION Network 28: Step-26
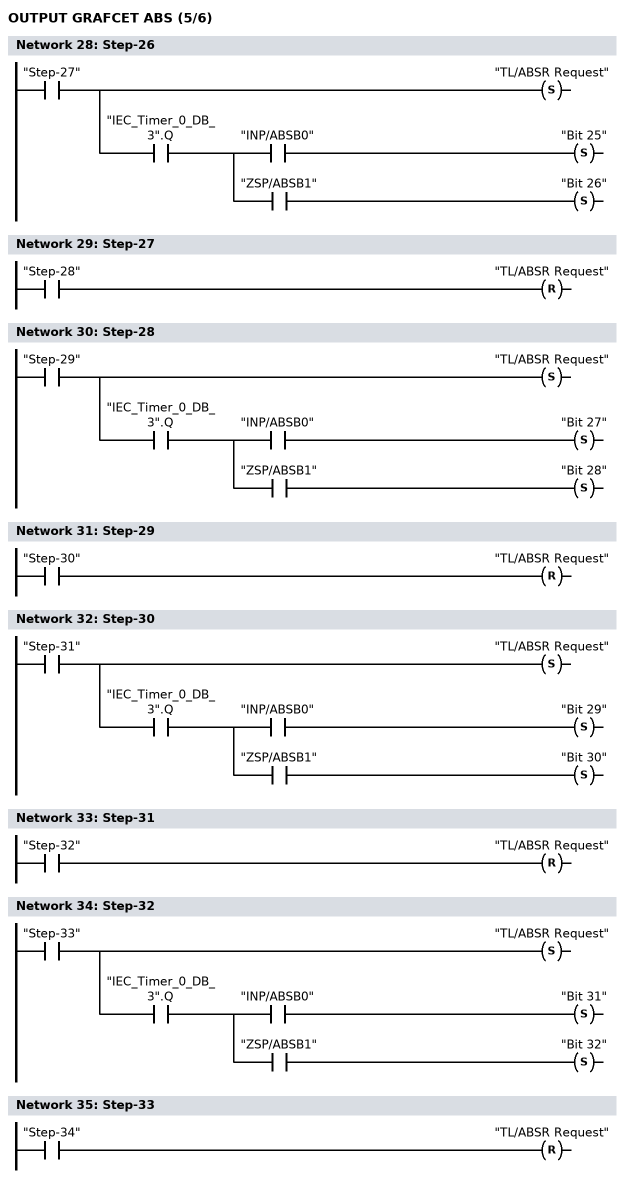
   RUNG wire#powerrail
      Contact( "Step-27" )
      wire#w1
      S_Coil( "TL/ABSR Request" )
   END_RUNG
   RUNG wire#w1
      Contact( "IEC_Timer_0_DB_3".Q )
      wire#w2
      Contact( "INP/ABSB0" )
      S_Coil( "Bit 25" )
   END_RUNG
   RUNG wire#w2
      Contact( "ZSP/ABSB1" )
      S_Coil( "Bit 26" )
   END_RUNG
   // the same network as SCL:
   IF "Step-27" THEN "TL/ABSR Request" := TRUE; END_IF;
   #_w1 := "Step-27" AND "IEC_Timer_0_DB_3".Q;
   IF #_w1 AND "INP/ABSB0" THEN "Bit 25" := TRUE; END_IF;
   IF #_w1 AND "ZSP/ABSB1" THEN "Bit 26" := TRUE; END_IF;
END_REGION

REGION Network 29: Step-27
   RUNG wire#powerrail
      Contact( "Step-28" )
      R_Coil( "TL/ABSR Request" )
   END_RUNG
   // the same network as SCL:
   IF "Step-28" THEN "TL/ABSR Request" := FALSE; END_IF;
END_REGION

REGION Network 30: Step-28
   RUNG wire#powerrail
      Contact( "Step-29" )
      wire#w1
      S_Coil( "TL/ABSR Request" )
   END_RUNG
   RUNG wire#w1
      Contact( "IEC_Timer_0_DB_3".Q )
      wire#w2
      Contact( "INP/ABSB0" )
      S_Coil( "Bit 27" )
   END_RUNG
   RUNG wire#w2
      Contact( "ZSP/ABSB1" )
      S_Coil( "Bit 28" )
   END_RUNG
   // the same network as SCL:
   IF "Step-29" THEN "TL/ABSR Request" := TRUE; END_IF;
   #_w1 := "Step-29" AND "IEC_Timer_0_DB_3".Q;
   IF #_w1 AND "INP/ABSB0" THEN "Bit 27" := TRUE; END_IF;
   IF #_w1 AND "ZSP/ABSB1" THEN "Bit 28" := TRUE; END_IF;
END_REGION

REGION Network 31: Step-29
   RUNG wire#powerrail
      Contact( "Step-30" )
      R_Coil( "TL/ABSR Request" )
   END_RUNG
   // the same network as SCL:
   IF "Step-30" THEN "TL/ABSR Request" := FALSE; END_IF;
END_REGION

REGION Network 32: Step-30
   RUNG wire#powerrail
      Contact( "Step-31" )
      wire#w1
      S_Coil( "TL/ABSR Request" )
   END_RUNG
   RUNG wire#w1
      Contact( "IEC_Timer_0_DB_3".Q )
      wire#w2
      Contact( "INP/ABSB0" )
      S_Coil( "Bit 29" )
   END_RUNG
   RUNG wire#w2
      Contact( "ZSP/ABSB1" )
      S_Coil( "Bit 30" )
   END_RUNG
   // the same network as SCL:
   IF "Step-31" THEN "TL/ABSR Request" := TRUE; END_IF;
   #_w1 := "Step-31" AND "IEC_Timer_0_DB_3".Q;
   IF #_w1 AND "INP/ABSB0" THEN "Bit 29" := TRUE; END_IF;
   IF #_w1 AND "ZSP/ABSB1" THEN "Bit 30" := TRUE; END_IF;
END_REGION

REGION Network 33: Step-31
   RUNG wire#powerrail
      Contact( "Step-32" )
      R_Coil( "TL/ABSR Request" )
   END_RUNG
   // the same network as SCL:
   IF "Step-32" THEN "TL/ABSR Request" := FALSE; END_IF;
END_REGION

REGION Network 34: Step-32
   RUNG wire#powerrail
      Contact( "Step-33" )
      wire#w1
      S_Coil( "TL/ABSR Request" )
   END_RUNG
   RUNG wire#w1
      Contact( "IEC_Timer_0_DB_3".Q )
      wire#w2
      Contact( "INP/ABSB0" )
      S_Coil( "Bit 31" )
   END_RUNG
   RUNG wire#w2
      Contact( "ZSP/ABSB1" )
      S_Coil( "Bit 32" )
   END_RUNG
   // the same network as SCL:
   IF "Step-33" THEN "TL/ABSR Request" := TRUE; END_IF;
   #_w1 := "Step-33" AND "IEC_Timer_0_DB_3".Q;
   IF #_w1 AND "INP/ABSB0" THEN "Bit 31" := TRUE; END_IF;
   IF #_w1 AND "ZSP/ABSB1" THEN "Bit 32" := TRUE; END_IF;
END_REGION

REGION Network 35: Step-33
   RUNG wire#powerrail
      Contact( "Step-34" )
      R_Coil( "TL/ABSR Request" )
   END_RUNG
   // the same network as SCL:
   IF "Step-34" THEN "TL/ABSR Request" := FALSE; END_IF;
END_REGION

REGION Network 36: Step-34
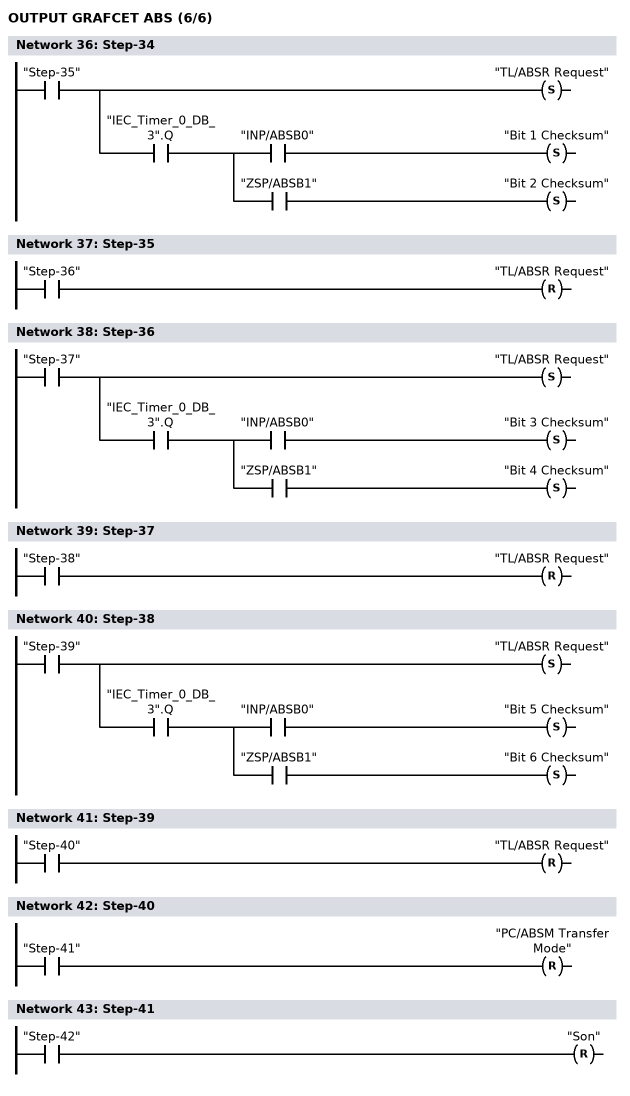
   RUNG wire#powerrail
      Contact( "Step-35" )
      wire#w1
      S_Coil( "TL/ABSR Request" )
   END_RUNG
   RUNG wire#w1
      Contact( "IEC_Timer_0_DB_3".Q )
      wire#w2
      Contact( "INP/ABSB0" )
      S_Coil( "Bit 1 Checksum" )
   END_RUNG
   RUNG wire#w2
      Contact( "ZSP/ABSB1" )
      S_Coil( "Bit 2 Checksum" )
   END_RUNG
   // the same network as SCL:
   IF "Step-35" THEN "TL/ABSR Request" := TRUE; END_IF;
   #_w1 := "Step-35" AND "IEC_Timer_0_DB_3".Q;
   IF #_w1 AND "INP/ABSB0" THEN "Bit 1 Checksum" := TRUE; END_IF;
   IF #_w1 AND "ZSP/ABSB1" THEN "Bit 2 Checksum" := TRUE; END_IF;
END_REGION

REGION Network 37: Step-35
   RUNG wire#powerrail
      Contact( "Step-36" )
      R_Coil( "TL/ABSR Request" )
   END_RUNG
   // the same network as SCL:
   IF "Step-36" THEN "TL/ABSR Request" := FALSE; END_IF;
END_REGION

REGION Network 38: Step-36
   RUNG wire#powerrail
      Contact( "Step-37" )
      wire#w1
      S_Coil( "TL/ABSR Request" )
   END_RUNG
   RUNG wire#w1
      Contact( "IEC_Timer_0_DB_3".Q )
      wire#w2
      Contact( "INP/ABSB0" )
      S_Coil( "Bit 3 Checksum" )
   END_RUNG
   RUNG wire#w2
      Contact( "ZSP/ABSB1" )
      S_Coil( "Bit 4 Checksum" )
   END_RUNG
   // the same network as SCL:
   IF "Step-37" THEN "TL/ABSR Request" := TRUE; END_IF;
   #_w1 := "Step-37" AND "IEC_Timer_0_DB_3".Q;
   IF #_w1 AND "INP/ABSB0" THEN "Bit 3 Checksum" := TRUE; END_IF;
   IF #_w1 AND "ZSP/ABSB1" THEN "Bit 4 Checksum" := TRUE; END_IF;
END_REGION

REGION Network 39: Step-37
   RUNG wire#powerrail
      Contact( "Step-38" )
      R_Coil( "TL/ABSR Request" )
   END_RUNG
   // the same network as SCL:
   IF "Step-38" THEN "TL/ABSR Request" := FALSE; END_IF;
END_REGION

REGION Network 40: Step-38
   RUNG wire#powerrail
      Contact( "Step-39" )
      wire#w1
      S_Coil( "TL/ABSR Request" )
   END_RUNG
   RUNG wire#w1
      Contact( "IEC_Timer_0_DB_3".Q )
      wire#w2
      Contact( "INP/ABSB0" )
      S_Coil( "Bit 5 Checksum" )
   END_RUNG
   RUNG wire#w2
      Contact( "ZSP/ABSB1" )
      S_Coil( "Bit 6 Checksum" )
   END_RUNG
   // the same network as SCL:
   IF "Step-39" THEN "TL/ABSR Request" := TRUE; END_IF;
   #_w1 := "Step-39" AND "IEC_Timer_0_DB_3".Q;
   IF #_w1 AND "INP/ABSB0" THEN "Bit 5 Checksum" := TRUE; END_IF;
   IF #_w1 AND "ZSP/ABSB1" THEN "Bit 6 Checksum" := TRUE; END_IF;
END_REGION

REGION Network 41: Step-39
   RUNG wire#powerrail
      Contact( "Step-40" )
      R_Coil( "TL/ABSR Request" )
   END_RUNG
   // the same network as SCL:
   IF "Step-40" THEN "TL/ABSR Request" := FALSE; END_IF;
END_REGION

REGION Network 42: Step-40
   RUNG wire#powerrail
      Contact( "Step-41" )
      R_Coil( "PC/ABSM Transfer Mode" )
   END_RUNG
   // the same network as SCL:
   IF "Step-41" THEN "PC/ABSM Transfer Mode" := FALSE; END_IF;
END_REGION

REGION Network 43: Step-41
   RUNG wire#powerrail
      Contact( "Step-42" )
      R_Coil( "Son" )
   END_RUNG
   // the same network as SCL:
   IF "Step-42" THEN "Son" := FALSE; END_IF;
END_REGION
END_FUNCTION

FUNCTION "AXIS CONTROL" : Void   // FC3, LAD
{ S7_Optimized_Access := 'TRUE' }
VERSION : 0.1
BEGIN

REGION Network 1
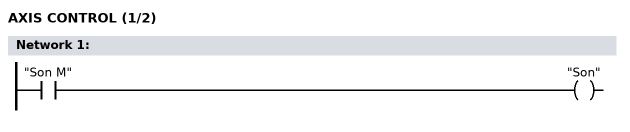
   RUNG wire#powerrail
      Contact( "Son M" )
      Coil( "Son" )
   END_RUNG
   // the same network as SCL:
   "Son" := "Son M";
END_REGION

REGION Network 2
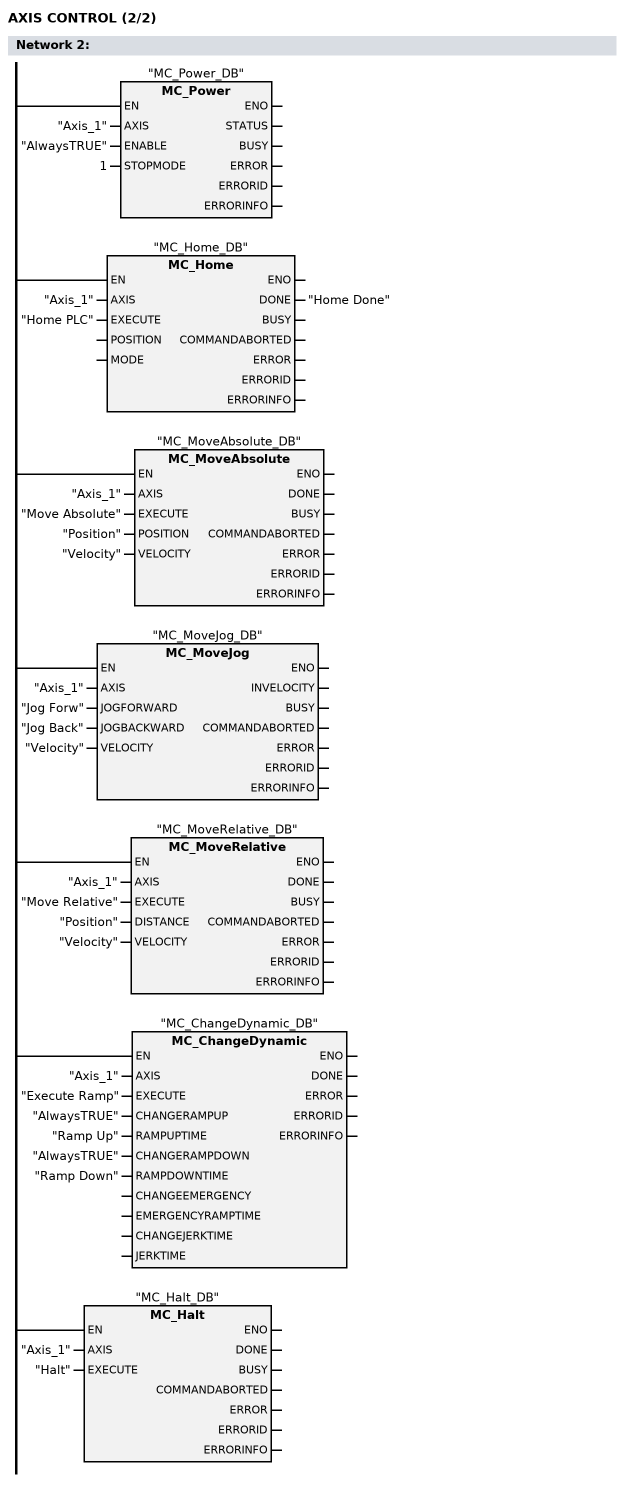
   "MC_Power_DB"(Axis := "Axis_1", Enable := "AlwaysTRUE", StopMode := 1);   // MC_Power
   "MC_Home_DB"(Axis := "Axis_1", Execute := "Home PLC", Done => "Home Done");   // MC_Home
   "MC_MoveAbsolute_DB"(Axis := "Axis_1",   // MC_MoveAbsolute
                        Execute := "Move Absolute",
                        Position := "Position",
                        Velocity := "Velocity");
   "MC_MoveJog_DB"(Axis := "Axis_1",   // MC_MoveJog
                   JogForward := "Jog Forw",
                   JogBackward := "Jog Back",
                   Velocity := "Velocity");
   "MC_MoveRelative_DB"(Axis := "Axis_1",   // MC_MoveRelative
                        Execute := "Move Relative",
                        Distance := "Position",
                        Velocity := "Velocity");
   "MC_ChangeDynamic_DB"(Axis := "Axis_1",   // MC_ChangeDynamic
                         Execute := "Execute Ramp",
                         ChangeRampUp := "AlwaysTRUE",
                         RampUpTime := "Ramp Up",
                         ChangeRampDown := "AlwaysTRUE",
                         RampDownTime := "Ramp Down");
   "MC_Halt_DB"(Axis := "Axis_1", Execute := "Halt");   // MC_Halt
END_REGION
END_FUNCTION

FUNCTION "LASERS CONTROL" : Void   // FC4, LAD
{ S7_Optimized_Access := 'TRUE' }
VERSION : 0.1
BEGIN

REGION Network 1
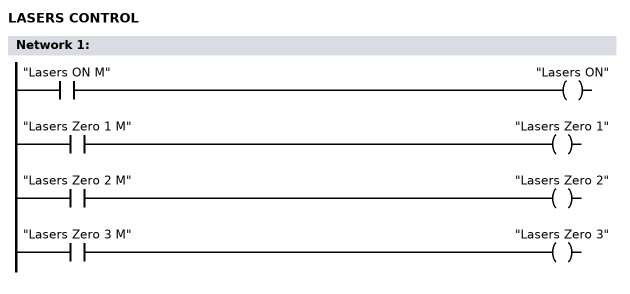
   RUNG wire#powerrail
      Contact( "Lasers ON M" )
      Coil( "Lasers ON" )
   END_RUNG
   RUNG wire#powerrail
      Contact( "Lasers Zero 1 M" )
      Coil( "Lasers Zero 1" )
   END_RUNG
   RUNG wire#powerrail
      Contact( "Lasers Zero 2 M" )
      Coil( "Lasers Zero 2" )
   END_RUNG
   RUNG wire#powerrail
      Contact( "Lasers Zero 3 M" )
      Coil( "Lasers Zero 3" )
   END_RUNG
   // the same network as SCL:
   "Lasers ON" := "Lasers ON M";
   "Lasers Zero 1" := "Lasers Zero 1 M";
   "Lasers Zero 2" := "Lasers Zero 2 M";
   "Lasers Zero 3" := "Lasers Zero 3 M";
END_REGION
END_FUNCTION

FUNCTION "BOT. PNEU. ACT. HOME" : Void   // FC5, LAD
{ S7_Optimized_Access := 'TRUE' }
VERSION : 0.1
BEGIN

REGION Network 1
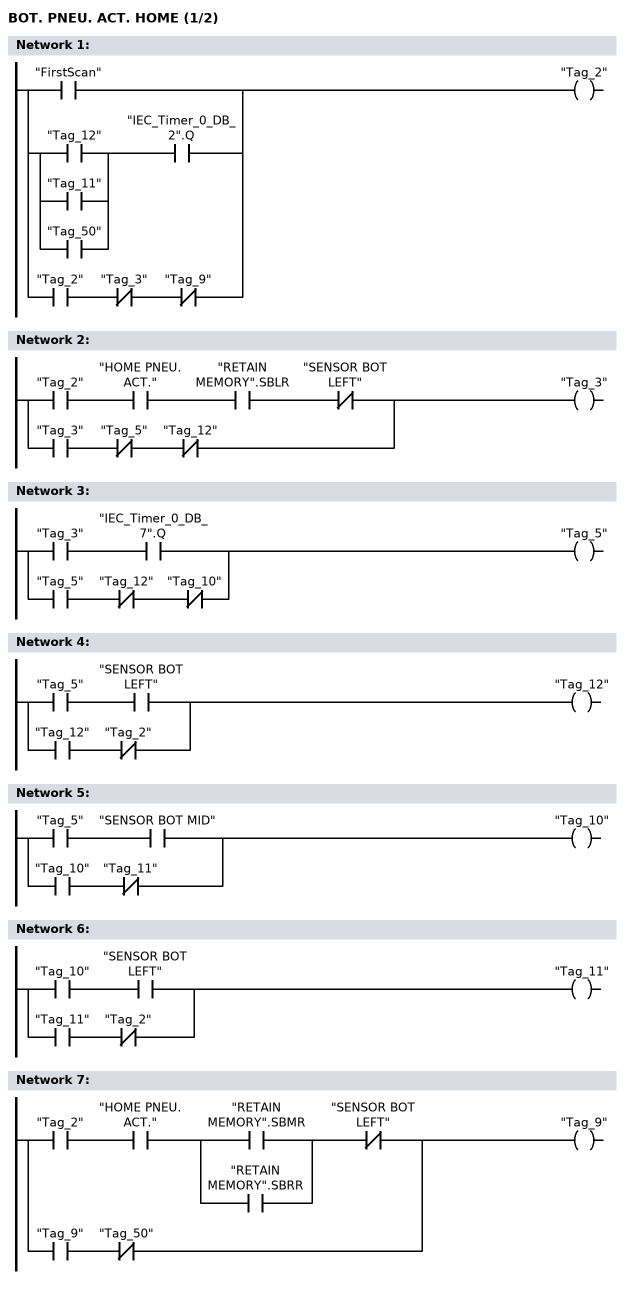
   RUNG wire#powerrail
      Contact( "FirstScan" )
      wire#w1
      Coil( "Tag_2" )
   END_RUNG
   RUNG wire#powerrail
      Contact( "Tag_12" )
      wire#w2
      Contact( "IEC_Timer_0_DB_2".Q )
   END_RUNG wire#w1
   RUNG wire#powerrail
      Contact( "Tag_11" )
   END_RUNG wire#w2
   RUNG wire#powerrail
      Contact( "Tag_50" )
   END_RUNG wire#w2
   RUNG wire#powerrail
      Contact( "Tag_2" )
      I_Contact( "Tag_3" )
      I_Contact( "Tag_9" )
   END_RUNG wire#w1
   // the same network as SCL:
   "Tag_2" := "FirstScan" OR (("Tag_12" OR "Tag_11" OR "Tag_50") AND "IEC_Timer_0_DB_2".Q) OR ("Tag_2" AND NOT "Tag_3" AND NOT "Tag_9");
END_REGION

REGION Network 2
   RUNG wire#powerrail
      Contact( "Tag_2" )
      Contact( "HOME PNEU. ACT." )
      Contact( "RETAIN MEMORY".SBLR )
      I_Contact( "SENSOR BOT LEFT" )
      wire#w1
      Coil( "Tag_3" )
   END_RUNG
   RUNG wire#powerrail
      Contact( "Tag_3" )
      I_Contact( "Tag_5" )
      I_Contact( "Tag_12" )
   END_RUNG wire#w1
   // the same network as SCL:
   "Tag_3" := ("Tag_2" AND "HOME PNEU. ACT." AND "RETAIN MEMORY".SBLR AND NOT "SENSOR BOT LEFT") OR ("Tag_3" AND NOT "Tag_5" AND NOT "Tag_12");
END_REGION

REGION Network 3
   RUNG wire#powerrail
      Contact( "Tag_3" )
      Contact( "IEC_Timer_0_DB_7".Q )
      wire#w1
      Coil( "Tag_5" )
   END_RUNG
   RUNG wire#powerrail
      Contact( "Tag_5" )
      I_Contact( "Tag_12" )
      I_Contact( "Tag_10" )
   END_RUNG wire#w1
   // the same network as SCL:
   "Tag_5" := ("Tag_3" AND "IEC_Timer_0_DB_7".Q) OR ("Tag_5" AND NOT "Tag_12" AND NOT "Tag_10");
END_REGION

REGION Network 4
   RUNG wire#powerrail
      Contact( "Tag_5" )
      Contact( "SENSOR BOT LEFT" )
      wire#w1
      Coil( "Tag_12" )
   END_RUNG
   RUNG wire#powerrail
      Contact( "Tag_12" )
      I_Contact( "Tag_2" )
   END_RUNG wire#w1
   // the same network as SCL:
   "Tag_12" := ("Tag_5" AND "SENSOR BOT LEFT") OR ("Tag_12" AND NOT "Tag_2");
END_REGION

REGION Network 5
   RUNG wire#powerrail
      Contact( "Tag_5" )
      Contact( "SENSOR BOT MID" )
      wire#w1
      Coil( "Tag_10" )
   END_RUNG
   RUNG wire#powerrail
      Contact( "Tag_10" )
      I_Contact( "Tag_11" )
   END_RUNG wire#w1
   // the same network as SCL:
   "Tag_10" := ("Tag_5" AND "SENSOR BOT MID") OR ("Tag_10" AND NOT "Tag_11");
END_REGION

REGION Network 6
   RUNG wire#powerrail
      Contact( "Tag_10" )
      Contact( "SENSOR BOT LEFT" )
      wire#w1
      Coil( "Tag_11" )
   END_RUNG
   RUNG wire#powerrail
      Contact( "Tag_11" )
      I_Contact( "Tag_2" )
   END_RUNG wire#w1
   // the same network as SCL:
   "Tag_11" := ("Tag_10" AND "SENSOR BOT LEFT") OR ("Tag_11" AND NOT "Tag_2");
END_REGION

REGION Network 7
   RUNG wire#powerrail
      Contact( "Tag_2" )
      Contact( "HOME PNEU. ACT." )
      wire#w1
      Contact( "RETAIN MEMORY".SBMR )
      wire#w2
      I_Contact( "SENSOR BOT LEFT" )
      wire#w3
      Coil( "Tag_9" )
   END_RUNG
   RUNG wire#w1
      Contact( "RETAIN MEMORY".SBRR )
   END_RUNG wire#w2
   RUNG wire#powerrail
      Contact( "Tag_9" )
      I_Contact( "Tag_50" )
   END_RUNG wire#w3
   // the same network as SCL:
   "Tag_9" := ("Tag_2" AND "HOME PNEU. ACT." AND ("RETAIN MEMORY".SBMR OR "RETAIN MEMORY".SBRR) AND NOT "SENSOR BOT LEFT") OR ("Tag_9" AND NOT "Tag_50");
END_REGION

REGION Network 8
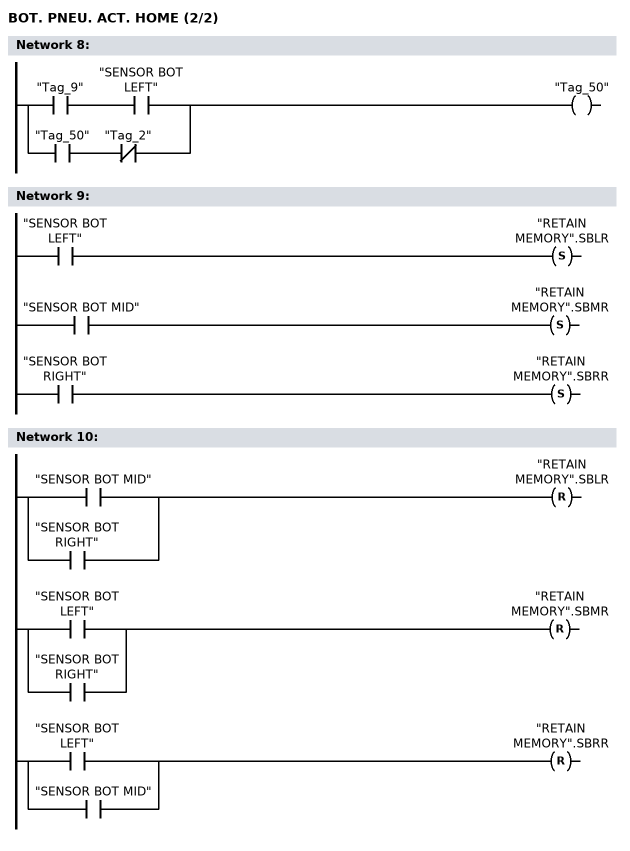
   RUNG wire#powerrail
      Contact( "Tag_9" )
      Contact( "SENSOR BOT LEFT" )
      wire#w1
      Coil( "Tag_50" )
   END_RUNG
   RUNG wire#powerrail
      Contact( "Tag_50" )
      I_Contact( "Tag_2" )
   END_RUNG wire#w1
   // the same network as SCL:
   "Tag_50" := ("Tag_9" AND "SENSOR BOT LEFT") OR ("Tag_50" AND NOT "Tag_2");
END_REGION

REGION Network 9
   RUNG wire#powerrail
      Contact( "SENSOR BOT LEFT" )
      S_Coil( "RETAIN MEMORY".SBLR )
   END_RUNG
   RUNG wire#powerrail
      Contact( "SENSOR BOT MID" )
      S_Coil( "RETAIN MEMORY".SBMR )
   END_RUNG
   RUNG wire#powerrail
      Contact( "SENSOR BOT RIGHT" )
      S_Coil( "RETAIN MEMORY".SBRR )
   END_RUNG
   // the same network as SCL:
   IF "SENSOR BOT LEFT" THEN "RETAIN MEMORY".SBLR := TRUE; END_IF;
   IF "SENSOR BOT MID" THEN "RETAIN MEMORY".SBMR := TRUE; END_IF;
   IF "SENSOR BOT RIGHT" THEN "RETAIN MEMORY".SBRR := TRUE; END_IF;
END_REGION

REGION Network 10
   RUNG wire#powerrail
      Contact( "SENSOR BOT MID" )
      wire#w1
      R_Coil( "RETAIN MEMORY".SBLR )
   END_RUNG
   RUNG wire#powerrail
      Contact( "SENSOR BOT RIGHT" )
   END_RUNG wire#w1
   RUNG wire#powerrail
      Contact( "SENSOR BOT LEFT" )
      wire#w2
      R_Coil( "RETAIN MEMORY".SBMR )
   END_RUNG
   RUNG wire#powerrail
      Contact( "SENSOR BOT RIGHT" )
   END_RUNG wire#w2
   RUNG wire#powerrail
      Contact( "SENSOR BOT LEFT" )
      wire#w3
      R_Coil( "RETAIN MEMORY".SBRR )
   END_RUNG
   RUNG wire#powerrail
      Contact( "SENSOR BOT MID" )
   END_RUNG wire#w3
   // the same network as SCL:
   IF "SENSOR BOT MID" OR "SENSOR BOT RIGHT" THEN "RETAIN MEMORY".SBLR := FALSE; END_IF;
   IF "SENSOR BOT LEFT" OR "SENSOR BOT RIGHT" THEN "RETAIN MEMORY".SBMR := FALSE; END_IF;
   IF "SENSOR BOT LEFT" OR "SENSOR BOT MID" THEN "RETAIN MEMORY".SBRR := FALSE; END_IF;
END_REGION
END_FUNCTION

FUNCTION "MODBUS SERVER" : Void   // FC6, LAD
{ S7_Optimized_Access := 'TRUE' }
VERSION : 0.1
BEGIN

REGION Network 1
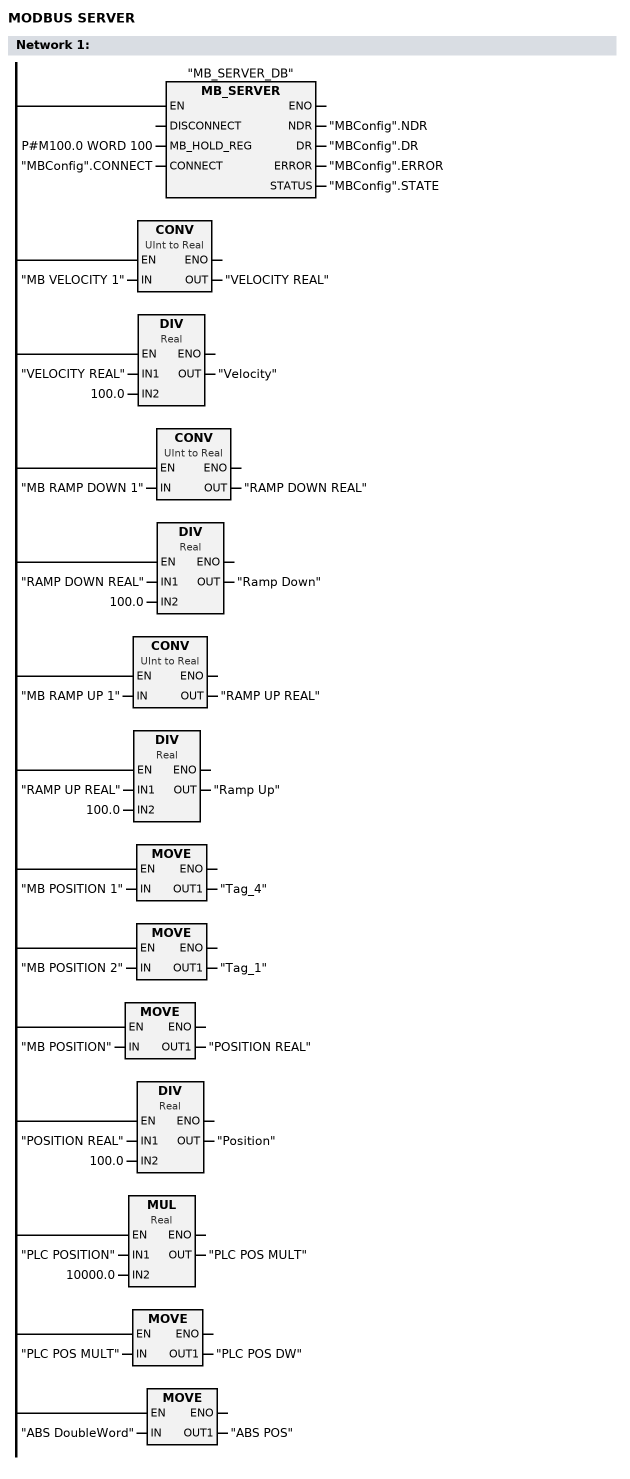
   "MB_SERVER_DB"(MB_HOLD_REG := P#M100.0 WORD 100,   // MB_SERVER
                  CONNECT := "MBConfig".CONNECT,
                  NDR => "MBConfig".NDR,
                  DR => "MBConfig".DR,
                  ERROR => "MBConfig".ERROR,
                  STATUS => "MBConfig".STATE);
   "VELOCITY REAL" := UINT_TO_REAL("MB VELOCITY 1");
   "Velocity" := "VELOCITY REAL" / 100.0;
   "RAMP DOWN REAL" := UINT_TO_REAL("MB RAMP DOWN 1");
   "Ramp Down" := "RAMP DOWN REAL" / 100.0;
   "RAMP UP REAL" := UINT_TO_REAL("MB RAMP UP 1");
   "Ramp Up" := "RAMP UP REAL" / 100.0;
   "Tag_4" := "MB POSITION 1";
   "Tag_1" := "MB POSITION 2";
   "POSITION REAL" := "MB POSITION";
   "Position" := "POSITION REAL" / 100.0;
   "PLC POS MULT" := "PLC POSITION" * 10000.0;
   "PLC POS DW" := "PLC POS MULT";
   "ABS POS" := "ABS DoubleWord";
END_REGION
END_FUNCTION

FUNCTION "BOT. PNEU. ACT. AUTO" : Void   // FC7, LAD
{ S7_Optimized_Access := 'TRUE' }
VERSION : 0.1
BEGIN

REGION Network 1
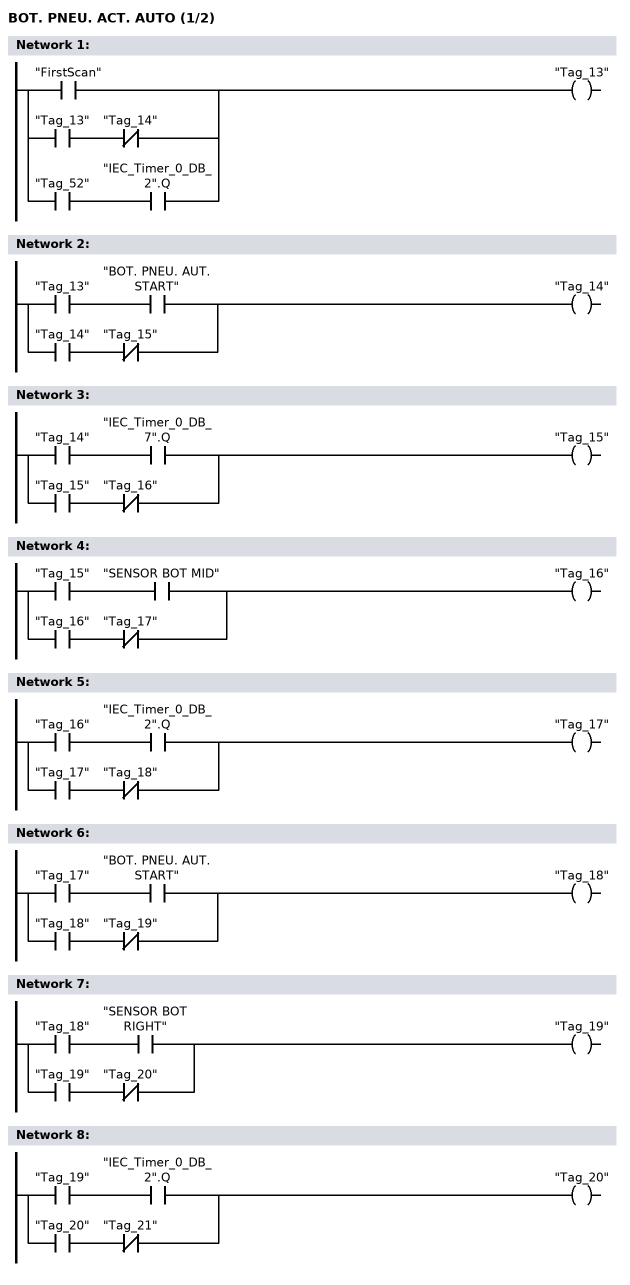
   RUNG wire#powerrail
      Contact( "FirstScan" )
      wire#w1
      Coil( "Tag_13" )
   END_RUNG
   RUNG wire#powerrail
      Contact( "Tag_13" )
      I_Contact( "Tag_14" )
   END_RUNG wire#w1
   RUNG wire#powerrail
      Contact( "Tag_52" )
      Contact( "IEC_Timer_0_DB_2".Q )
   END_RUNG wire#w1
   // the same network as SCL:
   "Tag_13" := "FirstScan" OR ("Tag_13" AND NOT "Tag_14") OR ("Tag_52" AND "IEC_Timer_0_DB_2".Q);
END_REGION

REGION Network 2
   RUNG wire#powerrail
      Contact( "Tag_13" )
      Contact( "BOT. PNEU. AUT. START" )
      wire#w1
      Coil( "Tag_14" )
   END_RUNG
   RUNG wire#powerrail
      Contact( "Tag_14" )
      I_Contact( "Tag_15" )
   END_RUNG wire#w1
   // the same network as SCL:
   "Tag_14" := ("Tag_13" AND "BOT. PNEU. AUT. START") OR ("Tag_14" AND NOT "Tag_15");
END_REGION

REGION Network 3
   RUNG wire#powerrail
      Contact( "Tag_14" )
      Contact( "IEC_Timer_0_DB_7".Q )
      wire#w1
      Coil( "Tag_15" )
   END_RUNG
   RUNG wire#powerrail
      Contact( "Tag_15" )
      I_Contact( "Tag_16" )
   END_RUNG wire#w1
   // the same network as SCL:
   "Tag_15" := ("Tag_14" AND "IEC_Timer_0_DB_7".Q) OR ("Tag_15" AND NOT "Tag_16");
END_REGION

REGION Network 4
   RUNG wire#powerrail
      Contact( "Tag_15" )
      Contact( "SENSOR BOT MID" )
      wire#w1
      Coil( "Tag_16" )
   END_RUNG
   RUNG wire#powerrail
      Contact( "Tag_16" )
      I_Contact( "Tag_17" )
   END_RUNG wire#w1
   // the same network as SCL:
   "Tag_16" := ("Tag_15" AND "SENSOR BOT MID") OR ("Tag_16" AND NOT "Tag_17");
END_REGION

REGION Network 5
   RUNG wire#powerrail
      Contact( "Tag_16" )
      Contact( "IEC_Timer_0_DB_2".Q )
      wire#w1
      Coil( "Tag_17" )
   END_RUNG
   RUNG wire#powerrail
      Contact( "Tag_17" )
      I_Contact( "Tag_18" )
   END_RUNG wire#w1
   // the same network as SCL:
   "Tag_17" := ("Tag_16" AND "IEC_Timer_0_DB_2".Q) OR ("Tag_17" AND NOT "Tag_18");
END_REGION

REGION Network 6
   RUNG wire#powerrail
      Contact( "Tag_17" )
      Contact( "BOT. PNEU. AUT. START" )
      wire#w1
      Coil( "Tag_18" )
   END_RUNG
   RUNG wire#powerrail
      Contact( "Tag_18" )
      I_Contact( "Tag_19" )
   END_RUNG wire#w1
   // the same network as SCL:
   "Tag_18" := ("Tag_17" AND "BOT. PNEU. AUT. START") OR ("Tag_18" AND NOT "Tag_19");
END_REGION

REGION Network 7
   RUNG wire#powerrail
      Contact( "Tag_18" )
      Contact( "SENSOR BOT RIGHT" )
      wire#w1
      Coil( "Tag_19" )
   END_RUNG
   RUNG wire#powerrail
      Contact( "Tag_19" )
      I_Contact( "Tag_20" )
   END_RUNG wire#w1
   // the same network as SCL:
   "Tag_19" := ("Tag_18" AND "SENSOR BOT RIGHT") OR ("Tag_19" AND NOT "Tag_20");
END_REGION

REGION Network 8
   RUNG wire#powerrail
      Contact( "Tag_19" )
      Contact( "IEC_Timer_0_DB_2".Q )
      wire#w1
      Coil( "Tag_20" )
   END_RUNG
   RUNG wire#powerrail
      Contact( "Tag_20" )
      I_Contact( "Tag_21" )
   END_RUNG wire#w1
   // the same network as SCL:
   "Tag_20" := ("Tag_19" AND "IEC_Timer_0_DB_2".Q) OR ("Tag_20" AND NOT "Tag_21");
END_REGION

REGION Network 9
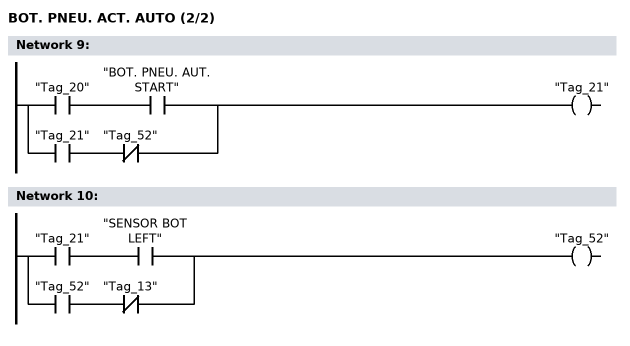
   RUNG wire#powerrail
      Contact( "Tag_20" )
      Contact( "BOT. PNEU. AUT. START" )
      wire#w1
      Coil( "Tag_21" )
   END_RUNG
   RUNG wire#powerrail
      Contact( "Tag_21" )
      I_Contact( "Tag_52" )
   END_RUNG wire#w1
   // the same network as SCL:
   "Tag_21" := ("Tag_20" AND "BOT. PNEU. AUT. START") OR ("Tag_21" AND NOT "Tag_52");
END_REGION

REGION Network 10
   RUNG wire#powerrail
      Contact( "Tag_21" )
      Contact( "SENSOR BOT LEFT" )
      wire#w1
      Coil( "Tag_52" )
   END_RUNG
   RUNG wire#powerrail
      Contact( "Tag_52" )
      I_Contact( "Tag_13" )
   END_RUNG wire#w1
   // the same network as SCL:
   "Tag_52" := ("Tag_21" AND "SENSOR BOT LEFT") OR ("Tag_52" AND NOT "Tag_13");
END_REGION
END_FUNCTION

FUNCTION "PNEU. ACT. OUTPUT" : Void   // FC8, LAD
{ S7_Optimized_Access := 'TRUE' }
VERSION : 0.1
BEGIN

REGION Network 1
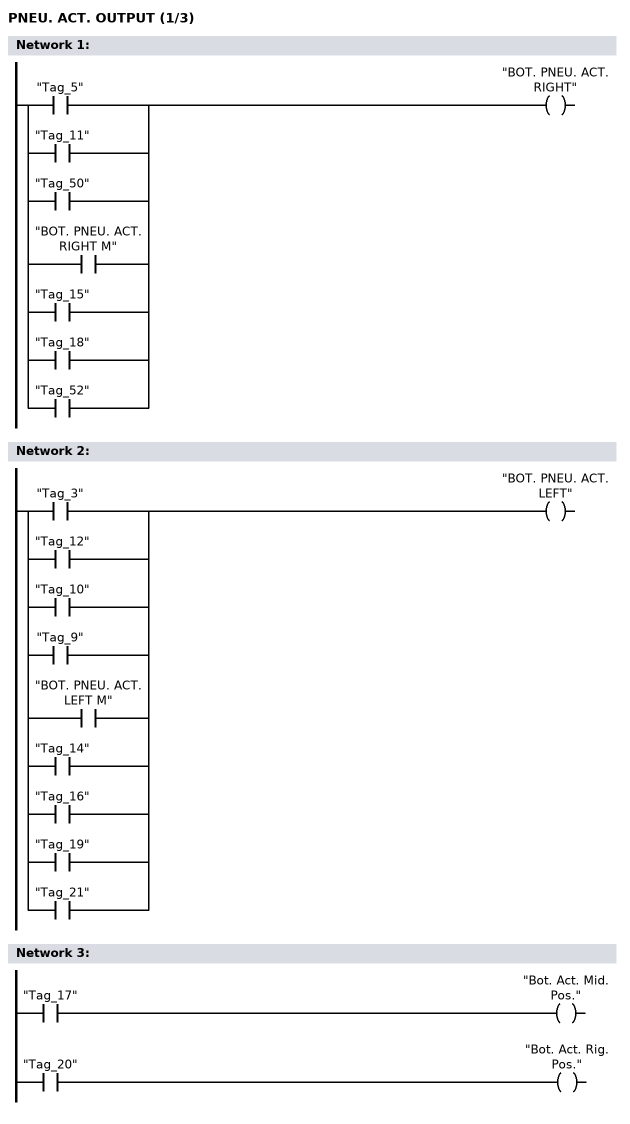
   RUNG wire#powerrail
      Contact( "Tag_5" )
      wire#w1
      Coil( "BOT. PNEU. ACT. RIGHT" )
   END_RUNG
   RUNG wire#powerrail
      Contact( "Tag_11" )
   END_RUNG wire#w1
   RUNG wire#powerrail
      Contact( "Tag_50" )
   END_RUNG wire#w1
   RUNG wire#powerrail
      Contact( "BOT. PNEU. ACT. RIGHT M" )
   END_RUNG wire#w1
   RUNG wire#powerrail
      Contact( "Tag_15" )
   END_RUNG wire#w1
   RUNG wire#powerrail
      Contact( "Tag_18" )
   END_RUNG wire#w1
   RUNG wire#powerrail
      Contact( "Tag_52" )
   END_RUNG wire#w1
   // the same network as SCL:
   "BOT. PNEU. ACT. RIGHT" := "Tag_5" OR "Tag_11" OR "Tag_50" OR "BOT. PNEU. ACT. RIGHT M" OR "Tag_15" OR "Tag_18" OR "Tag_52";
END_REGION

REGION Network 2
   RUNG wire#powerrail
      Contact( "Tag_3" )
      wire#w1
      Coil( "BOT. PNEU. ACT. LEFT" )
   END_RUNG
   RUNG wire#powerrail
      Contact( "Tag_12" )
   END_RUNG wire#w1
   RUNG wire#powerrail
      Contact( "Tag_10" )
   END_RUNG wire#w1
   RUNG wire#powerrail
      Contact( "Tag_9" )
   END_RUNG wire#w1
   RUNG wire#powerrail
      Contact( "BOT. PNEU. ACT. LEFT M" )
   END_RUNG wire#w1
   RUNG wire#powerrail
      Contact( "Tag_14" )
   END_RUNG wire#w1
   RUNG wire#powerrail
      Contact( "Tag_16" )
   END_RUNG wire#w1
   RUNG wire#powerrail
      Contact( "Tag_19" )
   END_RUNG wire#w1
   RUNG wire#powerrail
      Contact( "Tag_21" )
   END_RUNG wire#w1
   // the same network as SCL:
   "BOT. PNEU. ACT. LEFT" := "Tag_3" OR "Tag_12" OR "Tag_10" OR "Tag_9" OR "BOT. PNEU. ACT. LEFT M" OR "Tag_14" OR "Tag_16" OR "Tag_19" OR "Tag_21";
END_REGION

REGION Network 3
   RUNG wire#powerrail
      Contact( "Tag_17" )
      Coil( "Bot. Act. Mid. Pos." )
   END_RUNG
   RUNG wire#powerrail
      Contact( "Tag_20" )
      Coil( "Bot. Act. Rig. Pos." )
   END_RUNG
   // the same network as SCL:
   "Bot. Act. Mid. Pos." := "Tag_17";
   "Bot. Act. Rig. Pos." := "Tag_20";
END_REGION

REGION Network 4
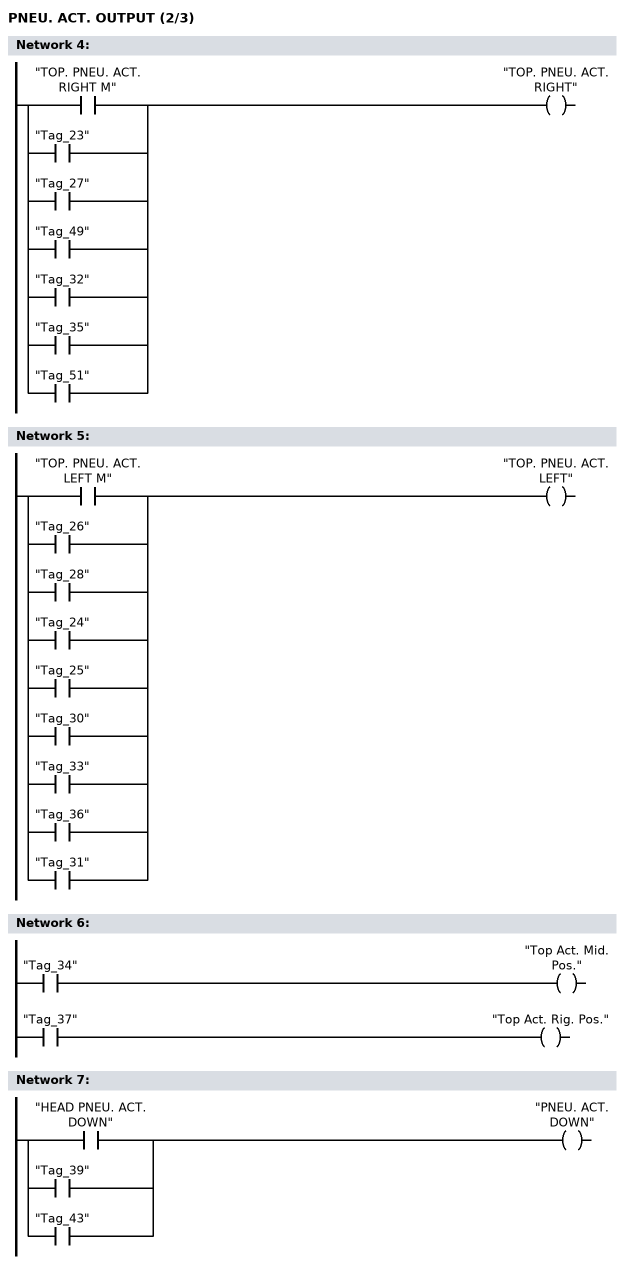
   RUNG wire#powerrail
      Contact( "TOP. PNEU. ACT. RIGHT M" )
      wire#w1
      Coil( "TOP. PNEU. ACT. RIGHT" )
   END_RUNG
   RUNG wire#powerrail
      Contact( "Tag_23" )
   END_RUNG wire#w1
   RUNG wire#powerrail
      Contact( "Tag_27" )
   END_RUNG wire#w1
   RUNG wire#powerrail
      Contact( "Tag_49" )
   END_RUNG wire#w1
   RUNG wire#powerrail
      Contact( "Tag_32" )
   END_RUNG wire#w1
   RUNG wire#powerrail
      Contact( "Tag_35" )
   END_RUNG wire#w1
   RUNG wire#powerrail
      Contact( "Tag_51" )
   END_RUNG wire#w1
   // the same network as SCL:
   "TOP. PNEU. ACT. RIGHT" := "TOP. PNEU. ACT. RIGHT M" OR "Tag_23" OR "Tag_27" OR "Tag_49" OR "Tag_32" OR "Tag_35" OR "Tag_51";
END_REGION

REGION Network 5
   RUNG wire#powerrail
      Contact( "TOP. PNEU. ACT. LEFT M" )
      wire#w1
      Coil( "TOP. PNEU. ACT. LEFT" )
   END_RUNG
   RUNG wire#powerrail
      Contact( "Tag_26" )
   END_RUNG wire#w1
   RUNG wire#powerrail
      Contact( "Tag_28" )
   END_RUNG wire#w1
   RUNG wire#powerrail
      Contact( "Tag_24" )
   END_RUNG wire#w1
   RUNG wire#powerrail
      Contact( "Tag_25" )
   END_RUNG wire#w1
   RUNG wire#powerrail
      Contact( "Tag_30" )
   END_RUNG wire#w1
   RUNG wire#powerrail
      Contact( "Tag_33" )
   END_RUNG wire#w1
   RUNG wire#powerrail
      Contact( "Tag_36" )
   END_RUNG wire#w1
   RUNG wire#powerrail
      Contact( "Tag_31" )
   END_RUNG wire#w1
   // the same network as SCL:
   "TOP. PNEU. ACT. LEFT" := "TOP. PNEU. ACT. LEFT M" OR "Tag_26" OR "Tag_28" OR "Tag_24" OR "Tag_25" OR "Tag_30" OR "Tag_33" OR "Tag_36" OR "Tag_31";
END_REGION

REGION Network 6
   RUNG wire#powerrail
      Contact( "Tag_34" )
      Coil( "Top Act. Mid. Pos." )
   END_RUNG
   RUNG wire#powerrail
      Contact( "Tag_37" )
      Coil( "Top Act. Rig. Pos." )
   END_RUNG
   // the same network as SCL:
   "Top Act. Mid. Pos." := "Tag_34";
   "Top Act. Rig. Pos." := "Tag_37";
END_REGION

REGION Network 7
   RUNG wire#powerrail
      Contact( "HEAD PNEU. ACT. DOWN" )
      wire#w1
      Coil( "PNEU. ACT. DOWN" )
   END_RUNG
   RUNG wire#powerrail
      Contact( "Tag_39" )
   END_RUNG wire#w1
   RUNG wire#powerrail
      Contact( "Tag_43" )
   END_RUNG wire#w1
   // the same network as SCL:
   "PNEU. ACT. DOWN" := "HEAD PNEU. ACT. DOWN" OR "Tag_39" OR "Tag_43";
END_REGION

REGION Network 8
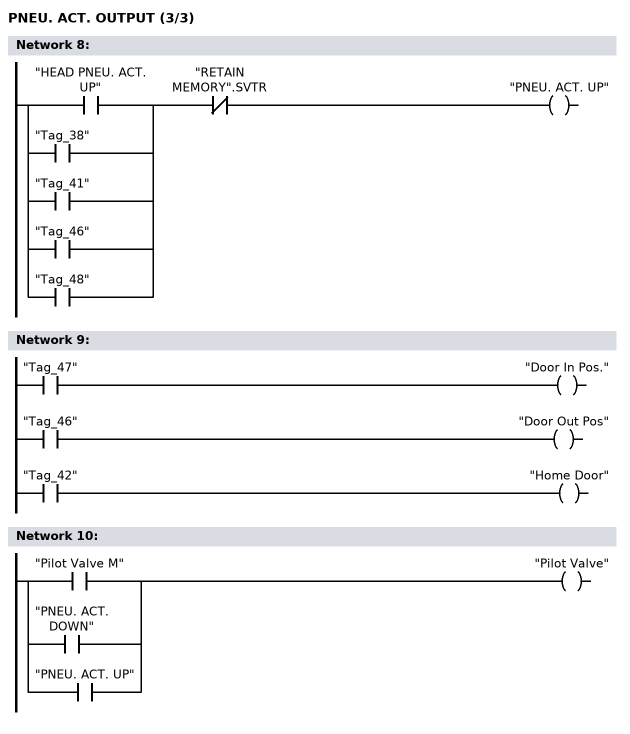
   RUNG wire#powerrail
      Contact( "HEAD PNEU. ACT. UP" )
      wire#w1
      I_Contact( "RETAIN MEMORY".SVTR )
      Coil( "PNEU. ACT. UP" )
   END_RUNG
   RUNG wire#powerrail
      Contact( "Tag_38" )
   END_RUNG wire#w1
   RUNG wire#powerrail
      Contact( "Tag_41" )
   END_RUNG wire#w1
   RUNG wire#powerrail
      Contact( "Tag_46" )
   END_RUNG wire#w1
   RUNG wire#powerrail
      Contact( "Tag_48" )
   END_RUNG wire#w1
   // the same network as SCL:
   "PNEU. ACT. UP" := ("HEAD PNEU. ACT. UP" OR "Tag_38" OR "Tag_41" OR "Tag_46" OR "Tag_48") AND NOT "RETAIN MEMORY".SVTR;
END_REGION

REGION Network 9
   RUNG wire#powerrail
      Contact( "Tag_47" )
      Coil( "Door In Pos." )
   END_RUNG
   RUNG wire#powerrail
      Contact( "Tag_46" )
      Coil( "Door Out Pos" )
   END_RUNG
   RUNG wire#powerrail
      Contact( "Tag_42" )
      Coil( "Home Door" )
   END_RUNG
   // the same network as SCL:
   "Door In Pos." := "Tag_47";
   "Door Out Pos" := "Tag_46";
   "Home Door" := "Tag_42";
END_REGION

REGION Network 10
   RUNG wire#powerrail
      Contact( "Pilot Valve M" )
      wire#w1
      Coil( "Pilot Valve" )
   END_RUNG
   RUNG wire#powerrail
      Contact( "PNEU. ACT. DOWN" )
   END_RUNG wire#w1
   RUNG wire#powerrail
      Contact( "PNEU. ACT. UP" )
   END_RUNG wire#w1
   // the same network as SCL:
   "Pilot Valve" := "Pilot Valve M" OR "PNEU. ACT. DOWN" OR "PNEU. ACT. UP";
END_REGION
END_FUNCTION

FUNCTION "PNEU. ACT. TIMERS" : Void   // FC9, LAD
{ S7_Optimized_Access := 'TRUE' }
VERSION : 0.1
BEGIN

REGION Network 1
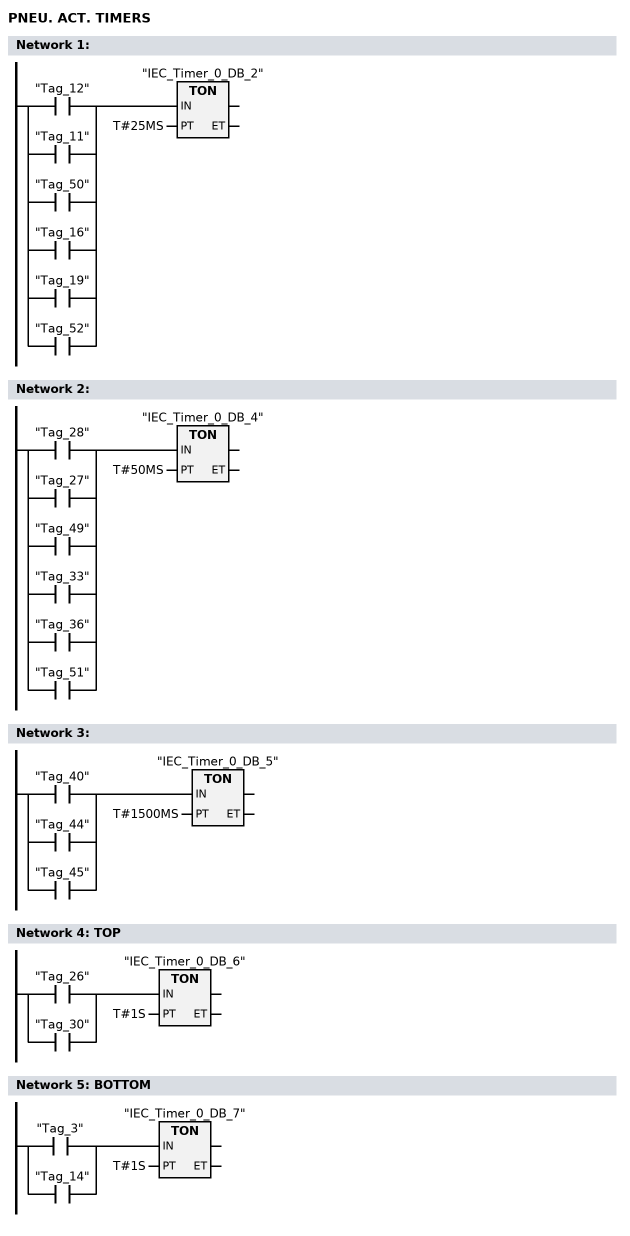
   "IEC_Timer_0_DB_2".TON(IN := "Tag_12" OR "Tag_11" OR "Tag_50" OR "Tag_16" OR "Tag_19" OR "Tag_52",
                          PT := T#25MS);
END_REGION

REGION Network 2
   "IEC_Timer_0_DB_4".TON(IN := "Tag_28" OR "Tag_27" OR "Tag_49" OR "Tag_33" OR "Tag_36" OR "Tag_51",
                          PT := T#50MS);
END_REGION

REGION Network 3
   "IEC_Timer_0_DB_5".TON(IN := "Tag_40" OR "Tag_44" OR "Tag_45", PT := T#1500MS);
END_REGION

REGION Network 4: TOP
   "IEC_Timer_0_DB_6".TON(IN := "Tag_26" OR "Tag_30", PT := T#1S);
END_REGION

REGION Network 5: BOTTOM
   "IEC_Timer_0_DB_7".TON(IN := "Tag_3" OR "Tag_14", PT := T#1S);
END_REGION
END_FUNCTION

FUNCTION "TOP PNEU. ACT. HOME" : Void   // FC10, LAD
{ S7_Optimized_Access := 'TRUE' }
VERSION : 0.1
BEGIN

REGION Network 1
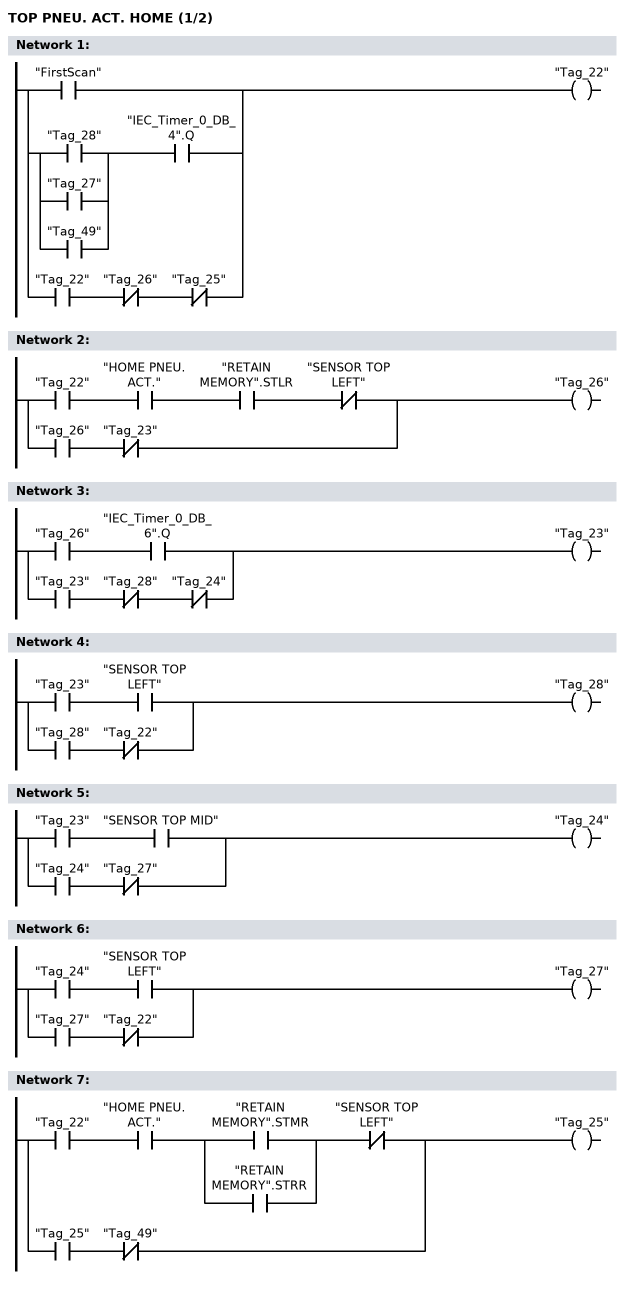
   RUNG wire#powerrail
      Contact( "FirstScan" )
      wire#w1
      Coil( "Tag_22" )
   END_RUNG
   RUNG wire#powerrail
      Contact( "Tag_28" )
      wire#w2
      Contact( "IEC_Timer_0_DB_4".Q )
   END_RUNG wire#w1
   RUNG wire#powerrail
      Contact( "Tag_27" )
   END_RUNG wire#w2
   RUNG wire#powerrail
      Contact( "Tag_49" )
   END_RUNG wire#w2
   RUNG wire#powerrail
      Contact( "Tag_22" )
      I_Contact( "Tag_26" )
      I_Contact( "Tag_25" )
   END_RUNG wire#w1
   // the same network as SCL:
   "Tag_22" := "FirstScan" OR (("Tag_28" OR "Tag_27" OR "Tag_49") AND "IEC_Timer_0_DB_4".Q) OR ("Tag_22" AND NOT "Tag_26" AND NOT "Tag_25");
END_REGION

REGION Network 2
   RUNG wire#powerrail
      Contact( "Tag_22" )
      Contact( "HOME PNEU. ACT." )
      Contact( "RETAIN MEMORY".STLR )
      I_Contact( "SENSOR TOP LEFT" )
      wire#w1
      Coil( "Tag_26" )
   END_RUNG
   RUNG wire#powerrail
      Contact( "Tag_26" )
      I_Contact( "Tag_23" )
   END_RUNG wire#w1
   // the same network as SCL:
   "Tag_26" := ("Tag_22" AND "HOME PNEU. ACT." AND "RETAIN MEMORY".STLR AND NOT "SENSOR TOP LEFT") OR ("Tag_26" AND NOT "Tag_23");
END_REGION

REGION Network 3
   RUNG wire#powerrail
      Contact( "Tag_26" )
      Contact( "IEC_Timer_0_DB_6".Q )
      wire#w1
      Coil( "Tag_23" )
   END_RUNG
   RUNG wire#powerrail
      Contact( "Tag_23" )
      I_Contact( "Tag_28" )
      I_Contact( "Tag_24" )
   END_RUNG wire#w1
   // the same network as SCL:
   "Tag_23" := ("Tag_26" AND "IEC_Timer_0_DB_6".Q) OR ("Tag_23" AND NOT "Tag_28" AND NOT "Tag_24");
END_REGION

REGION Network 4
   RUNG wire#powerrail
      Contact( "Tag_23" )
      Contact( "SENSOR TOP LEFT" )
      wire#w1
      Coil( "Tag_28" )
   END_RUNG
   RUNG wire#powerrail
      Contact( "Tag_28" )
      I_Contact( "Tag_22" )
   END_RUNG wire#w1
   // the same network as SCL:
   "Tag_28" := ("Tag_23" AND "SENSOR TOP LEFT") OR ("Tag_28" AND NOT "Tag_22");
END_REGION

REGION Network 5
   RUNG wire#powerrail
      Contact( "Tag_23" )
      Contact( "SENSOR TOP MID" )
      wire#w1
      Coil( "Tag_24" )
   END_RUNG
   RUNG wire#powerrail
      Contact( "Tag_24" )
      I_Contact( "Tag_27" )
   END_RUNG wire#w1
   // the same network as SCL:
   "Tag_24" := ("Tag_23" AND "SENSOR TOP MID") OR ("Tag_24" AND NOT "Tag_27");
END_REGION

REGION Network 6
   RUNG wire#powerrail
      Contact( "Tag_24" )
      Contact( "SENSOR TOP LEFT" )
      wire#w1
      Coil( "Tag_27" )
   END_RUNG
   RUNG wire#powerrail
      Contact( "Tag_27" )
      I_Contact( "Tag_22" )
   END_RUNG wire#w1
   // the same network as SCL:
   "Tag_27" := ("Tag_24" AND "SENSOR TOP LEFT") OR ("Tag_27" AND NOT "Tag_22");
END_REGION

REGION Network 7
   RUNG wire#powerrail
      Contact( "Tag_22" )
      Contact( "HOME PNEU. ACT." )
      wire#w1
      Contact( "RETAIN MEMORY".STMR )
      wire#w2
      I_Contact( "SENSOR TOP LEFT" )
      wire#w3
      Coil( "Tag_25" )
   END_RUNG
   RUNG wire#w1
      Contact( "RETAIN MEMORY".STRR )
   END_RUNG wire#w2
   RUNG wire#powerrail
      Contact( "Tag_25" )
      I_Contact( "Tag_49" )
   END_RUNG wire#w3
   // the same network as SCL:
   "Tag_25" := ("Tag_22" AND "HOME PNEU. ACT." AND ("RETAIN MEMORY".STMR OR "RETAIN MEMORY".STRR) AND NOT "SENSOR TOP LEFT") OR ("Tag_25" AND NOT "Tag_49");
END_REGION

REGION Network 8
